LIN {X 0,Y 411.211,Z 404.262,A -85,B 0,C 180,E1 -10479.728,E2 -10479.728} C_VEL
LIN {X 0,Y 411.171,Z 404.269,A -85,B 0,C 180,E1 -10483.134,E2 -10483.134} C_VEL
LIN {X 0,Y 411.171,Z 404.27,A -85,B 0,C 180,E1 -10485.881,E2 -10485.881} C_VEL
LIN {X 0,Y 411.213,Z 404.285,A -85,B 0,C 180,E1 -10487.705,E2 -10487.705} C_VEL
LIN {X 0,Y 411.99,Z 408.991,A -85,B 0,C 180,E1 -10490.864,E2 -10490.864} C_VEL
LIN {X 0,Y 412.564,Z 413.025,A -85,B 0,C 180,E1 -10493.401,E2 -10493.401} C_VEL
LIN {X 0,Y 412.538,Z 417.134,A -85,B 0,C 180,E1 -10495.793,E2 -10495.793} C_VEL
LIN {X 0,Y 412.031,Z 423.342,A -85,B 0,C 180,E1 -10499.223,E2 -10499.223} C_VEL
LIN {X 0,Y 411.473,Z 429.833,A -85,B 0,C 180,E1 -10502.644,E2 -10502.644} C_VEL
LIN {X 0,Y 411.104,Z 435.991,A -85,B 0,C 180,E1 -10505.777,E2 -10505.777} C_VEL
LIN {X 0,Y 410.797,Z 442.38,A -85,B 0,C 180,E1 -10508.945,E2 -10508.945} C_VEL
LIN {X 0,Y 410.522,Z 449.14,A -85,B 0,C 180,E1 -10512.118,E2 -10512.118} C_VEL
LIN {X 0,Y 413.255,Z 462.27,A -85,B 0,C 180,E1 -10512.668,E2 -10512.668} C_VEL
LIN {X 0,Y 414.885,Z 474.445,A -85,B 0,C 180,E1 -10513.327,E2 -10513.327} C_VEL
LIN {X 0,Y 415.191,Z 479.769,A -85,B 0,C 180,E1 -10513.656,E2 -10513.656} C_VEL
LIN {X 0,Y 414.353,Z 492.016,A -85,B 0,C 180,E1 -10514.506,E2 -10514.506} C_VEL
LIN {X 0,Y 413.49,Z 502.748,A -85,B 0,C 180,E1 -10515.457,E2 -10515.457} C_VEL
LIN {X 0,Y 412.834,Z 511.902,A -85,B 0,C 180,E1 -10516.463,E2 -10516.463} C_VEL
LIN {X 0,Y 412.087,Z 521.077,A -85,B 0,C 180,E1 -10517.691,E2 -10517.691} C_VEL
LIN {X 0,Y 411.228,Z 530.022,A -85,B 0,C 180,E1 -10519.164,E2 -10519.164} C_VEL
LIN {X 0,Y 410.717,Z 537.242,A -85,B 0,C 180,E1 -10520.645,E2 -10520.645} C_VEL
LIN {X 0,Y 410.354,Z 543.03,A -85,B 0,C 180,E1 -10522.125,E2 -10522.125} C_VEL
LIN {X 0,Y 410.045,Z 548.033,A -85,B 0,C 180,E1 -10523.774,E2 -10523.774} C_VEL
LIN {X 0,Y 410.024,Z 551.083,A -85,B 0,C 180,E1 -10525.084,E2 -10525.084} C_VEL
LIN {X 0,Y 409.935,Z 552.834,A -85,B 0,C 180,E1 -10526.068,E2 -10526.068} C_VEL
LIN {X 0,Y 409.967,Z 555.121,A -85,B 0,C 180,E1 -10528.035,E2 -10528.035} C_VEL
LIN {X 0,Y 409.936,Z 555.676,A -85,B 0,C 180,E1 -10529.017,E2 -10529.017} C_VEL
LIN {X 0,Y 409.926,Z 555.798,A -85,B 0,C 180,E1 -10530,E2 -10530} C_VEL
LIN {X 0,Y 409.967,Z 554.868,A -85,B 0,C 180,E1 -10531.965,E2 -10531.965} C_VEL
LIN {X 0,Y 409.929,Z 553.816,A -85,B 0,C 180,E1 -10532.948,E2 -10532.948} C_VEL
LIN {X 0,Y 409.935,Z 552.312,A -85,B 0,C 180,E1 -10533.932,E2 -10533.932} C_VEL
LIN {X 0,Y 410.025,Z 549.264,A -85,B 0,C 180,E1 -10535.409,E2 -10535.409} C_VEL
LIN {X 0,Y 410.167,Z 545.148,A -85,B 0,C 180,E1 -10536.888,E2 -10536.888} C_VEL
LIN {X 0,Y 410.488,Z 538.835,A -85,B 0,C 180,E1 -10538.616,E2 -10538.616} C_VEL
LIN {X 0,Y 410.916,Z 531.955,A -85,B 0,C 180,E1 -10540.096,E2 -10540.096} C_VEL
LIN {X 0,Y 411.365,Z 524.924,A -85,B 0,C 180,E1 -10541.33,E2 -10541.33} C_VEL
LIN {X 0,Y 412.025,Z 516.459,A -85,B 0,C 180,E1 -10542.561,E2 -10542.561} C_VEL
LIN {X 0,Y 412.68,Z 505.979,A -85,B 0,C 180,E1 -10543.793,E2 -10543.793} C_VEL
LIN {X 0,Y 413.431,Z 495.616,A -85,B 0,C 180,E1 -10544.772,E2 -10544.772} C_VEL
LIN {X 0,Y 414.099,Z 484.253,A -85,B 0,C 180,E1 -10545.63,E2 -10545.63} C_VEL
LIN {X 0,Y 414.498,Z 477.243,A -85,B 0,C 180,E1 -10546.056,E2 -10546.056} C_VEL
LIN {X 0,Y 412.757,Z 464.018,A -85,B 0,C 180,E1 -10546.759,E2 -10546.759} C_VEL
LIN {X 0,Y 410.638,Z 450.81,A -85,B 0,C 180,E1 -10547.267,E2 -10547.267} C_VEL
LIN {X 0,Y 410.406,Z 449.172,A -85,B 0,C 180,E1 -10547.314,E2 -10547.314} C_VEL
LIN {X 0,Y 410.705,Z 441.204,A -85,B 0,C 180,E1 -10551.06,E2 -10551.06} C_VEL
LIN {X 0,Y 410.962,Z 434.585,A -85,B 0,C 180,E1 -10554.231,E2 -10554.231} C_VEL
LIN {X 0,Y 411.272,Z 428.297,A -85,B 0,C 180,E1 -10557.302,E2 -10557.302} C_VEL
LIN {X 0,Y 411.717,Z 422.412,A -85,B 0,C 180,E1 -10560.235,E2 -10560.235} C_VEL
LIN {X 0,Y 412.033,Z 416.434,A -85,B 0,C 180,E1 -10563.302,E2 -10563.302} C_VEL
LIN {X 0,Y 412.291,Z 412.421,A -85,B 0,C 180,E1 -10565.419,E2 -10565.419} C_VEL
LIN {X 0,Y 411.848,Z 407.948,A -85,B 0,C 180,E1 -10567.902,E2 -10567.902} C_VEL
LIN {X 0,Y 411.242,Z 404.261,A -85,B 0,C 180,E1 -10570.083,E2 -10570.083} C_VEL
LIN {X 0,Y 411.215,Z 404.265,A -85,B 0,C 180,E1 -10573.127,E2 -10573.127} C_VEL
LIN {X 0,Y 411.173,Z 404.265,A -85,B 0,C 180,E1 -10575.879,E2 -10575.879} C_VEL
LIN {X 0,Y 411.16,Z 404.271,A -85,B 0,C 180,E1 -10578.771,E2 -10578.771} C_VEL
LIN {X 0,Y 411.195,Z 404.263,A -85,B 0,C 180,E1 -10582.026,E2 -10582.026} C_VEL
LIN {X 0,Y 411.201,Z 404.263,A -85,B 0,C 180,E1 -10585.666,E2 -10585.666} C_VEL
LIN {X 0,Y 411.192,Z 404.265,A -85,B 0,C 180,E1 -10589.152,E2 -10589.152} C_VEL
LIN {X 0,Y 411.253,Z 404.26,A -85,B 0,C 180,E1 -10592.522,E2 -10592.522} C_VEL
LIN {X 0,Y 411.22,Z 404.26,A -85,B 0,C 180,E1 -10595.784,E2 -10595.784} C_VEL
LIN {X 0,Y 411.189,Z 404.266,A -85,B 0,C 180,E1 -10598.965,E2 -10598.965} C_VEL
LIN {X 0,Y 411.245,Z 404.259,A -85,B 0,C 180,E1 -10602.084,E2 -10602.084} C_VEL
LIN {X 0,Y 411.251,Z 404.258,A -85,B 0,C 180,E1 -10605.147,E2 -10605.147} C_VEL
LIN {X 0,Y 411.276,Z 404.256,A -85,B 0,C 180,E1 -10608.167,E2 -10608.167} C_VEL
LIN {X 0,Y 411.474,Z 404.232,A -85,B 0,C 180,E1 -10612.146,E2 -10612.146} C_VEL
LIN {X 0,Y 411.482,Z 404.23,A -85,B 0,C 180,E1 -10614.118,E2 -10614.118} C_VEL
LIN {X 0,Y 411.506,Z 404.227,A -85,B 0,C 180,E1 -10618.042,E2 -10618.042} C_VEL
LIN {X 0,Y 411.635,Z 404.211,A -85,B 0,C 180,E1 -10620,E2 -10620} C_VEL
LIN {X 0,Y 411.46,Z 404.231,A -85,B 0,C 180,E1 -10622.937,E2 -10622.937} C_VEL
LIN {X 0,Y 411.453,Z 404.232,A -85,B 0,C 180,E1 -10626.867,E2 -10626.867} C_VEL
LIN {X 0,Y 411.286,Z 404.254,A -85,B 0,C 180,E1 -10629.839,E2 -10629.839} C_VEL
LIN {X 0,Y 411.304,Z 404.25,A -85,B 0,C 180,E1 -10633.109,E2 -10633.109} C_VEL
LIN {X 0,Y 411.249,Z 404.257,A -85,B 0,C 180,E1 -10636.889,E2 -10636.889} C_VEL
LIN {X 0,Y 411.222,Z 404.262,A -85,B 0,C 180,E1 -10639.987,E2 -10639.987} C_VEL
LIN {X 0,Y 411.196,Z 404.263,A -85,B 0,C 180,E1 -10643.148,E2 -10643.148} C_VEL
LIN {X 0,Y 411.23,Z 404.26,A -85,B 0,C 180,E1 -10646.381,E2 -10646.381} C_VEL
LIN {X 0,Y 411.204,Z 404.264,A -85,B 0,C 180,E1 -10649.712,E2 -10649.712} C_VEL
LIN {X 0,Y 411.2,Z 404.263,A -85,B 0,C 180,E1 -10653.156,E2 -10653.156} C_VEL
LIN {X 0,Y 411.189,Z 404.263,A -85,B 0,C 180,E1 -10656.554,E2 -10656.554} C_VEL
LIN {X 0,Y 411.223,Z 404.265,A -85,B 0,C 180,E1 -10659.731,E2 -10659.731} C_VEL
LIN {X 0,Y 411.226,Z 404.259,A -85,B 0,C 180,E1 -10663.127,E2 -10663.127} C_VEL
LIN {X 0,Y 411.226,Z 404.261,A -85,B 0,C 180,E1 -10665.873,E2 -10665.873} C_VEL
LIN {X 0,Y 411.205,Z 404.26,A -85,B 0,C 180,E1 -10668.765,E2 -10668.765} C_VEL
LIN {X 0,Y 411.201,Z 404.261,A -85,B 0,C 180,E1 -10672.028,E2 -10672.028} C_VEL
LIN {X 0,Y 411.203,Z 404.264,A -85,B 0,C 180,E1 -10675.667,E2 -10675.667} C_VEL
LIN {X 0,Y 411.187,Z 404.268,A -85,B 0,C 180,E1 -10679.153,E2 -10679.153} C_VEL
LIN {X 0,Y 411.257,Z 404.254,A -85,B 0,C 180,E1 -10682.523,E2 -10682.523} C_VEL
LIN {X 0,Y 411.216,Z 404.26,A -85,B 0,C 180,E1 -10685.785,E2 -10685.785} C_VEL
LIN {X 0,Y 411.119,Z 404.272,A -85,B 0,C 180,E1 -10687.909,E2 -10687.909} C_VEL
LIN {X 0,Y 411.038,Z 404.286,A -85,B 0,C 180,E1 -10688.958,E2 -10688.958} C_VEL
LIN {X 0,Y 411.028,Z 405.412,A -85,B 0,C 180,E1 -10690.122,E2 -10690.122} C_VEL
LIN {X 0,Y 410.929,Z 409.509,A -85,B 0,C 180,E1 -10693.285,E2 -10693.285} C_VEL
LIN {X 0,Y 410.805,Z 414.704,A -85,B 0,C 180,E1 -10697.199,E2 -10697.199} C_VEL
LIN {X 0,Y 410.584,Z 420.085,A -85,B 0,C 180,E1 -10701.138,E2 -10701.138} C_VEL
LIN {X 0,Y 410.621,Z 422.814,A -85,B 0,C 180,E1 -10703.119,E2 -10703.119} C_VEL
LIN {X 0,Y 410.429,Z 427.997,A -85,B 0,C 180,E1 -10706.779,E2 -10706.779} C_VEL
LIN {X 0,Y 412.935,Z 441.081,A -85,B 0,C 180,E1 -10707.302,E2 -10707.302} C_VEL
LIN {X 0,Y 414.936,Z 451.663,A -85,B 0,C 180,E1 -10707.877,E2 -10707.877} C_VEL
LIN {X 0,Y 414.296,Z 464.392,A -85,B 0,C 180,E1 -10708.664,E2 -10708.664} C_VEL
LIN {X 0,Y 413.609,Z 475.006,A -85,B 0,C 180,E1 -10709.513,E2 -10709.513} C_VEL
LIN {X 0,Y 412.859,Z 485.842,A -85,B 0,C 180,E1 -10710.61,E2 -10710.61} C_VEL
LIN {X 0,Y 412.21,Z 494.689,A -85,B 0,C 180,E1 -10711.71,E2 -10711.71} C_VEL
LIN {X 0,Y 411.455,Z 504.315,A -85,B 0,C 180,E1 -10713.182,E2 -10713.182} C_VEL
LIN {X 0,Y 410.935,Z 511.972,A -85,B 0,C 180,E1 -10714.66,E2 -10714.66} C_VEL
LIN {X 0,Y 410.607,Z 518.371,A -85,B 0,C 180,E1 -10716.209,E2 -10716.209} C_VEL
LIN {X 0,Y 410.256,Z 523.742,A -85,B 0,C 180,E1 -10717.877,E2 -10717.877} C_VEL
LIN {X 0,Y 410.049,Z 527.342,A -85,B 0,C 180,E1 -10719.371,E2 -10719.371} C_VEL
LIN {X 0,Y 409.956,Z 529.338,A -85,B 0,C 180,E1 -10720.511,E2 -10720.511} C_VEL
LIN {X 0,Y 409.264,Z 530.53,A -85,B 0,C 180,E1 -10721.315,E2 -10721.315} C_VEL
LIN {X 0,Y 406.302,Z 531.836,A -85,B 0,C 180,E1 -10722.632,E2 -10722.632} C_VEL
LIN {X 0,Y 403.811,Z 532.355,A -85,B 0,C 180,E1 -10723.704,E2 -10723.704} C_VEL
LIN {X 0,Y 402.763,Z 532.438,A -85,B 0,C 180,E1 -10724.536,E2 -10724.536} C_VEL
LIN {X 0,Y 402.69,Z 532.364,A -85,B 0,C 180,E1 -10724.818,E2 -10724.818} C_VEL
LIN {X 0,Y 402.765,Z 531.637,A -85,B 0,C 180,E1 -10726.319,E2 -10726.319} C_VEL
LIN {X 0,Y 402.899,Z 529.294,A -85,B 0,C 180,E1 -10728.299,E2 -10728.299} C_VEL
LIN {X 0,Y 403.167,Z 526.562,A -85,B 0,C 180,E1 -10729.725,E2 -10729.725} C_VEL
LIN {X 0,Y 403.5,Z 522.035,A -85,B 0,C 180,E1 -10731.455,E2 -10731.455} C_VEL
LIN {X 0,Y 404.058,Z 515.464,A -85,B 0,C 180,E1 -10733.311,E2 -10733.311} C_VEL
LIN {X 0,Y 404.681,Z 508.327,A -85,B 0,C 180,E1 -10734.883,E2 -10734.883} C_VEL
LIN {X 0,Y 405.391,Z 500.677,A -85,B 0,C 180,E1 -10736.236,E2 -10736.236} C_VEL
LIN {X 0,Y 406.193,Z 491.422,A -85,B 0,C 180,E1 -10737.57,E2 -10737.57} C_VEL
LIN {X 0,Y 407.089,Z 481.869,A -85,B 0,C 180,E1 -10738.686,E2 -10738.686} C_VEL
LIN {X 0,Y 407.925,Z 471.292,A -85,B 0,C 180,E1 -10739.691,E2 -10739.691} C_VEL
LIN {X 0,Y 408.762,Z 459.381,A -85,B 0,C 180,E1 -10740.573,E2 -10740.573} C_VEL
LIN {X 0,Y 409.008,Z 453.009,A -85,B 0,C 180,E1 -10740.961,E2 -10740.961} C_VEL
LIN {X 0,Y 406.66,Z 441.02,A -85,B 0,C 180,E1 -10741.685,E2 -10741.685} C_VEL
LIN {X 0,Y 403.291,Z 428.389,A -85,B 0,C 180,E1 -10742.323,E2 -10742.323} C_VEL
LIN {X 0,Y 403.46,Z 423.131,A -85,B 0,C 180,E1 -10746.317,E2 -10746.317} C_VEL
LIN {X 0,Y 403.621,Z 419.902,A -85,B 0,C 180,E1 -10748.817,E2 -10748.817} C_VEL
LIN {X 0,Y 403.788,Z 416.481,A -85,B 0,C 180,E1 -10751.546,E2 -10751.546} C_VEL
LIN {X 0,Y 403.953,Z 412.879,A -85,B 0,C 180,E1 -10754.494,E2 -10754.494} C_VEL
LIN {X 0,Y 404.163,Z 409.553,A -85,B 0,C 180,E1 -10757.299,E2 -10757.299} C_VEL
LIN {X 0,Y 404.226,Z 406.491,A -85,B 0,C 180,E1 -10759.962,E2 -10759.962} C_VEL
LIN {X 0,Y 404.131,Z 405.148,A -85,B 0,C 180,E1 -10761.241,E2 -10761.241} C_VEL
LIN {X 0,Y 404.181,Z 405.145,A -85,B 0,C 180,E1 -10764.984,E2 -10764.984} C_VEL
LIN {X 0,Y 404.144,Z 405.146,A -85,B 0,C 180,E1 -10768.554,E2 -10768.554} C_VEL
LIN {X 0,Y 404.193,Z 405.137,A -85,B 0,C 180,E1 -10772,E2 -10772} C_VEL
LIN {X 0,Y 404.169,Z 405.142,A -85,B 0,C 180,E1 -10775.334,E2 -10775.334} C_VEL
LIN {X 0,Y 404.132,Z 405.145,A -85,B 0,C 180,E1 -10778.58,E2 -10778.58} C_VEL
LIN {X 0,Y 404.204,Z 405.138,A -85,B 0,C 180,E1 -10781.762,E2 -10781.762} C_VEL
LIN {X 0,Y 404.2,Z 405.137,A -85,B 0,C 180,E1 -10784.882,E2 -10784.882} C_VEL
LIN {X 0,Y 404.251,Z 405.13,A -85,B 0,C 180,E1 -10787.958,E2 -10787.958} C_VEL
LIN {X 0,Y 404.427,Z 405.11,A -85,B 0,C 180,E1 -10792.1,E2 -10792.1} C_VEL
LIN {X 0,Y 404.418,Z 405.11,A -85,B 0,C 180,E1 -10794.015,E2 -10794.015} C_VEL
LIN {X 0,Y 404.477,Z 405.104,A -85,B 0,C 180,E1 -10798.009,E2 -10798.009} C_VEL
LIN {X 0,Y 404.605,Z 405.086,A -85,B 0,C 180,E1 -10800,E2 -10800} C_VEL
LIN {X 0,Y 404.419,Z 405.109,A -85,B 0,C 180,E1 -10802.989,E2 -10802.989} C_VEL
LIN {X 0,Y 404.401,Z 405.109,A -85,B 0,C 180,E1 -10806.988,E2 -10806.988} C_VEL
LIN {X 0,Y 404.266,Z 405.13,A -85,B 0,C 180,E1 -10810.012,E2 -10810.012} C_VEL
LIN {X 0,Y 404.261,Z 405.13,A -85,B 0,C 180,E1 -10813.212,E2 -10813.212} C_VEL
LIN {X 0,Y 404.214,Z 405.136,A -85,B 0,C 180,E1 -10817.009,E2 -10817.009} C_VEL
LIN {X 0,Y 404.159,Z 405.146,A -85,B 0,C 180,E1 -10820.352,E2 -10820.352} C_VEL
LIN {X 0,Y 404.165,Z 405.144,A -85,B 0,C 180,E1 -10823.575,E2 -10823.575} C_VEL
LIN {X 0,Y 404.179,Z 405.14,A -85,B 0,C 180,E1 -10825.767,E2 -10825.767} C_VEL
LIN {X 0,Y 404.194,Z 405.14,A -85,B 0,C 180,E1 -10828,E2 -10828} C_VEL
LIN {X 0,Y 404.139,Z 405.144,A -85,B 0,C 180,E1 -10831.559,E2 -10831.559} C_VEL
LIN {X 0,Y 404.182,Z 405.139,A -85,B 0,C 180,E1 -10835.017,E2 -10835.017} C_VEL
LIN {X 0,Y 404.153,Z 405.14,A -85,B 0,C 180,E1 -10838.757,E2 -10838.757} C_VEL
LIN {X 0,Y 404.12,Z 405.149,A -85,B 0,C 180,E1 -10841.6,E2 -10841.6} C_VEL
LIN {X 0,Y 404.145,Z 405.145,A -85,B 0,C 180,E1 -10844.523,E2 -10844.523} C_VEL
LIN {X 0,Y 404.184,Z 405.324,A -85,B 0,C 180,E1 -10847.444,E2 -10847.444} C_VEL
LIN {X 0,Y 404.876,Z 409.076,A -85,B 0,C 180,E1 -10850.04,E2 -10850.04} C_VEL
LIN {X 0,Y 405.507,Z 413.425,A -85,B 0,C 180,E1 -10852.868,E2 -10852.868} C_VEL
LIN {X 0,Y 405.597,Z 417.15,A -85,B 0,C 180,E1 -10855.124,E2 -10855.124} C_VEL
LIN {X 0,Y 405.078,Z 423.338,A -85,B 0,C 180,E1 -10858.635,E2 -10858.635} C_VEL
LIN {X 0,Y 404.634,Z 428.57,A -85,B 0,C 180,E1 -10861.469,E2 -10861.469} C_VEL
LIN {X 0,Y 404.116,Z 435.939,A -85,B 0,C 180,E1 -10865.331,E2 -10865.331} C_VEL
LIN {X 0,Y 403.725,Z 443.366,A -85,B 0,C 180,E1 -10869.093,E2 -10869.093} C_VEL
LIN {X 0,Y 403.452,Z 448.874,A -85,B 0,C 180,E1 -10871.74,E2 -10871.74} C_VEL
LIN {X 0,Y 406.317,Z 462.111,A -85,B 0,C 180,E1 -10872.315,E2 -10872.315} C_VEL
LIN {X 0,Y 407.968,Z 473.966,A -85,B 0,C 180,E1 -10872.971,E2 -10872.971} C_VEL
LIN {X 0,Y 408.401,Z 480.273,A -85,B 0,C 180,E1 -10873.376,E2 -10873.376} C_VEL
LIN {X 0,Y 407.55,Z 492.36,A -85,B 0,C 180,E1 -10874.241,E2 -10874.241} C_VEL
LIN {X 0,Y 406.64,Z 502.952,A -85,B 0,C 180,E1 -10875.206,E2 -10875.206} C_VEL
LIN {X 0,Y 405.934,Z 512.024,A -85,B 0,C 180,E1 -10876.228,E2 -10876.228} C_VEL
LIN {X 0,Y 405.144,Z 521.129,A -85,B 0,C 180,E1 -10877.477,E2 -10877.477} C_VEL
LIN {X 0,Y 404.224,Z 530.031,A -85,B 0,C 180,E1 -10878.974,E2 -10878.974} C_VEL
LIN {X 0,Y 403.686,Z 537.211,A -85,B 0,C 180,E1 -10880.48,E2 -10880.48} C_VEL
LIN {X 0,Y 403.299,Z 542.957,A -85,B 0,C 180,E1 -10881.986,E2 -10881.986} C_VEL
LIN {X 0,Y 402.958,Z 548.252,A -85,B 0,C 180,E1 -10883.795,E2 -10883.795} C_VEL
LIN {X 0,Y 402.937,Z 550.956,A -85,B 0,C 180,E1 -10884.997,E2 -10884.997} C_VEL
LIN {X 0,Y 402.855,Z 552.687,A -85,B 0,C 180,E1 -10885.998,E2 -10885.998} C_VEL
LIN {X 0,Y 402.865,Z 554.947,A -85,B 0,C 180,E1 -10888,E2 -10888} C_VEL
LIN {X 0,Y 402.863,Z 555.484,A -85,B 0,C 180,E1 -10889,E2 -10889} C_VEL
LIN {X 0,Y 402.851,Z 555.588,A -85,B 0,C 180,E1 -10890,E2 -10890} C_VEL
LIN {X 0,Y 402.863,Z 555.303,A -85,B 0,C 180,E1 -10890.999,E2 -10890.999} C_VEL
LIN {X 0,Y 402.88,Z 554.633,A -85,B 0,C 180,E1 -10891.999,E2 -10891.999} C_VEL
LIN {X 0,Y 402.829,Z 553.562,A -85,B 0,C 180,E1 -10893,E2 -10893} C_VEL
LIN {X 0,Y 402.855,Z 552.038,A -85,B 0,C 180,E1 -10894.001,E2 -10894.001} C_VEL
LIN {X 0,Y 402.926,Z 548.959,A -85,B 0,C 180,E1 -10895.505,E2 -10895.505} C_VEL
LIN {X 0,Y 403.081,Z 544.812,A -85,B 0,C 180,E1 -10897.01,E2 -10897.01} C_VEL
LIN {X 0,Y 403.424,Z 538.466,A -85,B 0,C 180,E1 -10898.768,E2 -10898.768} C_VEL
LIN {X 0,Y 403.862,Z 531.548,A -85,B 0,C 180,E1 -10900.274,E2 -10900.274} C_VEL
LIN {X 0,Y 404.383,Z 524.478,A -85,B 0,C 180,E1 -10901.529,E2 -10901.529} C_VEL
LIN {X 0,Y 405.033,Z 515.949,A -85,B 0,C 180,E1 -10902.781,E2 -10902.781} C_VEL
LIN {X 0,Y 405.748,Z 505.392,A -85,B 0,C 180,E1 -10904.033,E2 -10904.033} C_VEL
LIN {X 0,Y 406.593,Z 493.504,A -85,B 0,C 180,E1 -10905.155,E2 -10905.155} C_VEL
LIN {X 0,Y 407.346,Z 481.504,A -85,B 0,C 180,E1 -10906.024,E2 -10906.024} C_VEL
LIN {X 0,Y 407.408,Z 476.897,A -85,B 0,C 180,E1 -10906.308,E2 -10906.308} C_VEL
LIN {X 0,Y 405.69,Z 463.838,A -85,B 0,C 180,E1 -10907.015,E2 -10907.015} C_VEL
LIN {X 0,Y 403.618,Z 450.803,A -85,B 0,C 180,E1 -10907.524,E2 -10907.524} C_VEL
LIN {X 0,Y 403.344,Z 448.906,A -85,B 0,C 180,E1 -10907.609,E2 -10907.609} C_VEL
LIN {X 0,Y 403.656,Z 440.915,A -85,B 0,C 180,E1 -10911.446,E2 -10911.446} C_VEL
LIN {X 0,Y 403.936,Z 434.311,A -85,B 0,C 180,E1 -10914.681,E2 -10914.681} C_VEL
LIN {X 0,Y 404.287,Z 427.671,A -85,B 0,C 180,E1 -10917.992,E2 -10917.992} C_VEL
LIN {X 0,Y 404.826,Z 421.044,A -85,B 0,C 180,E1 -10921.386,E2 -10921.386} C_VEL
LIN {X 0,Y 405.197,Z 414.384,A -85,B 0,C 180,E1 -10924.915,E2 -10924.915} C_VEL
LIN {X 0,Y 405.065,Z 410.533,A -85,B 0,C 180,E1 -10927.049,E2 -10927.049} C_VEL
LIN {X 0,Y 404.217,Z 405.137,A -85,B 0,C 180,E1 -10930.206,E2 -10930.206} C_VEL
LIN {X 0,Y 404.19,Z 405.14,A -85,B 0,C 180,E1 -10933.089,E2 -10933.089} C_VEL
LIN {X 0,Y 404.152,Z 405.14,A -85,B 0,C 180,E1 -10935.926,E2 -10935.926} C_VEL
LIN {X 0,Y 404.115,Z 405.147,A -85,B 0,C 180,E1 -10938.634,E2 -10938.634} C_VEL
LIN {X 0,Y 404.152,Z 405.141,A -85,B 0,C 180,E1 -10941.491,E2 -10941.491} C_VEL
LIN {X 0,Y 404.18,Z 405.14,A -85,B 0,C 180,E1 -10944.983,E2 -10944.983} C_VEL
LIN {X 0,Y 404.14,Z 405.145,A -85,B 0,C 180,E1 -10948.553,E2 -10948.553} C_VEL
LIN {X 0,Y 404.192,Z 405.136,A -85,B 0,C 180,E1 -10952,E2 -10952} C_VEL
LIN {X 0,Y 404.17,Z 405.14,A -85,B 0,C 180,E1 -10955.334,E2 -10955.334} C_VEL
LIN {X 0,Y 404.131,Z 405.146,A -85,B 0,C 180,E1 -10958.58,E2 -10958.58} C_VEL
LIN {X 0,Y 404.202,Z 405.134,A -85,B 0,C 180,E1 -10961.761,E2 -10961.761} C_VEL
LIN {X 0,Y 404.198,Z 405.137,A -85,B 0,C 180,E1 -10964.881,E2 -10964.881} C_VEL
LIN {X 0,Y 404.248,Z 405.13,A -85,B 0,C 180,E1 -10967.958,E2 -10967.958} C_VEL
LIN {X 0,Y 404.425,Z 405.109,A -85,B 0,C 180,E1 -10972.099,E2 -10972.099} C_VEL
LIN {X 0,Y 404.428,Z 405.109,A -85,B 0,C 180,E1 -10974.015,E2 -10974.015} C_VEL
LIN {X 0,Y 404.475,Z 405.103,A -85,B 0,C 180,E1 -10978.008,E2 -10978.008} C_VEL
LIN {X 0,Y 404.605,Z 405.087,A -85,B 0,C 180,E1 -10980,E2 -10980} C_VEL
LIN {X 0,Y 404.417,Z 405.108,A -85,B 0,C 180,E1 -10982.988,E2 -10982.988} C_VEL
LIN {X 0,Y 404.404,Z 405.11,A -85,B 0,C 180,E1 -10986.987,E2 -10986.987} C_VEL
LIN {X 0,Y 404.252,Z 405.13,A -85,B 0,C 180,E1 -10990.012,E2 -10990.012} C_VEL
LIN {X 0,Y 404.258,Z 405.127,A -85,B 0,C 180,E1 -10993.211,E2 -10993.211} C_VEL
LIN {X 0,Y 404.207,Z 405.133,A -85,B 0,C 180,E1 -10997.007,E2 -10997.007} C_VEL
LIN {X 0,Y 404.156,Z 405.143,A -85,B 0,C 180,E1 -11000.352,E2 -11000.352} C_VEL
LIN {X 0,Y 404.162,Z 405.141,A -85,B 0,C 180,E1 -11003.575,E2 -11003.575} C_VEL
LIN {X 0,Y 404.176,Z 405.14,A -85,B 0,C 180,E1 -11005.767,E2 -11005.767} C_VEL
LIN {X 0,Y 404.19,Z 405.14,A -85,B 0,C 180,E1 -11008,E2 -11008} C_VEL
LIN {X 0,Y 404.139,Z 405.144,A -85,B 0,C 180,E1 -11011.56,E2 -11011.56} C_VEL
LIN {X 0,Y 404.179,Z 405.137,A -85,B 0,C 180,E1 -11015.017,E2 -11015.017} C_VEL
LIN {X 0,Y 404.158,Z 405.139,A -85,B 0,C 180,E1 -11018.756,E2 -11018.756} C_VEL
LIN {X 0,Y 404.186,Z 405.14,A -85,B 0,C 180,E1 -11021.611,E2 -11021.611} C_VEL
LIN {X 0,Y 404.196,Z 405.133,A -85,B 0,C 180,E1 -11024.531,E2 -11024.531} C_VEL
LIN {X 0,Y 404.202,Z 405.136,A -85,B 0,C 180,E1 -11027.306,E2 -11027.306} C_VEL
LIN {X 0,Y 404.164,Z 405.139,A -85,B 0,C 180,E1 -11029.956,E2 -11029.956} C_VEL
LIN {X 0,Y 404.137,Z 405.144,A -85,B 0,C 180,E1 -11033.125,E2 -11033.125} C_VEL
LIN {X 0,Y 404.142,Z 405.14,A -85,B 0,C 180,E1 -11036.188,E2 -11036.188} C_VEL
LIN {X 0,Y 404.143,Z 405.142,A -85,B 0,C 180,E1 -11039.716,E2 -11039.716} C_VEL
LIN {X 0,Y 404.194,Z 405.139,A -85,B 0,C 180,E1 -11043.124,E2 -11043.124} C_VEL
LIN {X 0,Y 404.171,Z 405.141,A -85,B 0,C 180,E1 -11045.335,E2 -11045.335} C_VEL
LIN {X 0,Y 404.128,Z 405.145,A -85,B 0,C 180,E1 -11047.506,E2 -11047.506} C_VEL
LIN {X 0,Y 404.009,Z 405.158,A -85,B 0,C 180,E1 -11048.574,E2 -11048.574} C_VEL
LIN {X 0,Y 403.97,Z 406.064,A -85,B 0,C 180,E1 -11049.96,E2 -11049.96} C_VEL
LIN {X 0,Y 403.866,Z 410.146,A -85,B 0,C 180,E1 -11053.156,E2 -11053.156} C_VEL
LIN {X 0,Y 403.748,Z 415.319,A -85,B 0,C 180,E1 -11057.106,E2 -11057.106} C_VEL
LIN {X 0,Y 403.508,Z 420.529,A -85,B 0,C 180,E1 -11060.982,E2 -11060.982} C_VEL
LIN {X 0,Y 403.559,Z 423.344,A -85,B 0,C 180,E1 -11063.052,E2 -11063.052} C_VEL
LIN {X 0,Y 403.363,Z 428.145,A -85,B 0,C 180,E1 -11066.504,E2 -11066.504} C_VEL
LIN {X 0,Y 406.235,Z 443.034,A -85,B 0,C 180,E1 -11067.136,E2 -11067.136} C_VEL
LIN {X 0,Y 407.965,Z 452.196,A -85,B 0,C 180,E1 -11067.654,E2 -11067.654} C_VEL
LIN {X 0,Y 407.431,Z 463.966,A -85,B 0,C 180,E1 -11068.394,E2 -11068.394} C_VEL
LIN {X 0,Y 406.705,Z 474.709,A -85,B 0,C 180,E1 -11069.258,E2 -11069.258} C_VEL
LIN {X 0,Y 405.954,Z 485.657,A -85,B 0,C 180,E1 -11070.372,E2 -11070.372} C_VEL
LIN {X 0,Y 405.23,Z 494.579,A -85,B 0,C 180,E1 -11071.491,E2 -11071.491} C_VEL
LIN {X 0,Y 404.448,Z 504.256,A -85,B 0,C 180,E1 -11072.988,E2 -11072.988} C_VEL
LIN {X 0,Y 403.893,Z 511.978,A -85,B 0,C 180,E1 -11074.491,E2 -11074.491} C_VEL
LIN {X 0,Y 403.572,Z 518.162,A -85,B 0,C 180,E1 -11075.998,E2 -11075.998} C_VEL
LIN {X 0,Y 403.263,Z 523.096,A -85,B 0,C 180,E1 -11077.511,E2 -11077.511} C_VEL
LIN {X 0,Y 402.996,Z 526.911,A -85,B 0,C 180,E1 -11079.03,E2 -11079.03} C_VEL
LIN {X 0,Y 402.849,Z 529.565,A -85,B 0,C 180,E1 -11080.5,E2 -11080.5} C_VEL
LIN {X 0,Y 402.812,Z 531.668,A -85,B 0,C 180,E1 -11082.299,E2 -11082.299} C_VEL
LIN {X 0,Y 402.688,Z 532.46,A -85,B 0,C 180,E1 -11084.143,E2 -11084.143} C_VEL
LIN {X 0,Y 402.69,Z 532.364,A -85,B 0,C 180,E1 -11084.818,E2 -11084.818} C_VEL
LIN {X 0,Y 402.062,Z 532.145,A -85,B 0,C 180,E1 -11085.654,E2 -11085.654} C_VEL
LIN {X 0,Y 399.272,Z 531.288,A -85,B 0,C 180,E1 -11087.012,E2 -11087.012} C_VEL
LIN {X 0,Y 396.953,Z 530.034,A -85,B 0,C 180,E1 -11088.096,E2 -11088.096} C_VEL
LIN {X 0,Y 396.029,Z 528.682,A -85,B 0,C 180,E1 -11088.922,E2 -11088.922} C_VEL
LIN {X 0,Y 395.994,Z 528.144,A -85,B 0,C 180,E1 -11089.197,E2 -11089.197} C_VEL
LIN {X 0,Y 396.289,Z 524.633,A -85,B 0,C 180,E1 -11090.774,E2 -11090.774} C_VEL
LIN {X 0,Y 396.682,Z 519.839,A -85,B 0,C 180,E1 -11092.39,E2 -11092.39} C_VEL
LIN {X 0,Y 397.245,Z 513.657,A -85,B 0,C 180,E1 -11094.011,E2 -11094.011} C_VEL
LIN {X 0,Y 397.902,Z 506.844,A -85,B 0,C 180,E1 -11095.446,E2 -11095.446} C_VEL
LIN {X 0,Y 398.793,Z 497.792,A -85,B 0,C 180,E1 -11096.987,E2 -11096.987} C_VEL
LIN {X 0,Y 399.635,Z 488.915,A -85,B 0,C 180,E1 -11098.204,E2 -11098.204} C_VEL
LIN {X 0,Y 400.692,Z 477.927,A -85,B 0,C 180,E1 -11099.413,E2 -11099.413} C_VEL
LIN {X 0,Y 401.552,Z 467.224,A -85,B 0,C 180,E1 -11100.356,E2 -11100.356} C_VEL
LIN {X 0,Y 402.342,Z 454.903,A -85,B 0,C 180,E1 -11101.199,E2 -11101.199} C_VEL
LIN {X 0,Y 399.971,Z 442.386,A -85,B 0,C 180,E1 -11101.99,E2 -11101.99} C_VEL
LIN {X 0,Y 396.213,Z 428.617,A -85,B 0,C 180,E1 -11102.716,E2 -11102.716} C_VEL
LIN {X 0,Y 396.353,Z 424.582,A -85,B 0,C 180,E1 -11105.813,E2 -11105.813} C_VEL
LIN {X 0,Y 396.58,Z 420.845,A -85,B 0,C 180,E1 -11108.763,E2 -11108.763} C_VEL
LIN {X 0,Y 396.789,Z 416.465,A -85,B 0,C 180,E1 -11112.303,E2 -11112.303} C_VEL
LIN {X 0,Y 396.948,Z 413.152,A -85,B 0,C 180,E1 -11115.088,E2 -11115.088} C_VEL
LIN {X 0,Y 397.158,Z 409.756,A -85,B 0,C 180,E1 -11118.005,E2 -11118.005} C_VEL
LIN {X 0,Y 397.164,Z 407.073,A -85,B 0,C 180,E1 -11120.429,E2 -11120.429} C_VEL
LIN {X 0,Y 397.088,Z 406.026,A -85,B 0,C 180,E1 -11121.723,E2 -11121.723} C_VEL
LIN {X 0,Y 397.121,Z 406.024,A -85,B 0,C 180,E1 -11125.506,E2 -11125.506} C_VEL
LIN {X 0,Y 397.082,Z 406.025,A -85,B 0,C 180,E1 -11129.118,E2 -11129.118} C_VEL
LIN {X 0,Y 397.19,Z 406.011,A -85,B 0,C 180,E1 -11132.61,E2 -11132.61} C_VEL
LIN {X 0,Y 397.123,Z 406.018,A -85,B 0,C 180,E1 -11135.981,E2 -11135.981} C_VEL
LIN {X 0,Y 397.133,Z 406.017,A -85,B 0,C 180,E1 -11139.705,E2 -11139.705} C_VEL
LIN {X 0,Y 397.176,Z 406.011,A -85,B 0,C 180,E1 -11142.845,E2 -11142.845} C_VEL
LIN {X 0,Y 397.223,Z 406.005,A -85,B 0,C 180,E1 -11146.703,E2 -11146.703} C_VEL
LIN {X 0,Y 397.213,Z 406.005,A -85,B 0,C 180,E1 -11149.809,E2 -11149.809} C_VEL
LIN {X 0,Y 397.358,Z 405.988,A -85,B 0,C 180,E1 -11152.888,E2 -11152.888} C_VEL
LIN {X 0,Y 397.249,Z 406.004,A -85,B 0,C 180,E1 -11154.925,E2 -11154.925} C_VEL
LIN {X 0,Y 397.446,Z 405.98,A -85,B 0,C 180,E1 -11157.973,E2 -11157.973} C_VEL
LIN {X 0,Y 397.574,Z 405.962,A -85,B 0,C 180,E1 -11160,E2 -11160} C_VEL
LIN {X 0,Y 397.377,Z 405.986,A -85,B 0,C 180,E1 -11163.042,E2 -11163.042} C_VEL
LIN {X 0,Y 397.369,Z 405.987,A -85,B 0,C 180,E1 -11166.092,E2 -11166.092} C_VEL
LIN {X 0,Y 397.252,Z 406.002,A -85,B 0,C 180,E1 -11169.162,E2 -11169.162} C_VEL
LIN {X 0,Y 397.225,Z 406.005,A -85,B 0,C 180,E1 -11172.258,E2 -11172.258} C_VEL
LIN {X 0,Y 397.181,Z 406.011,A -85,B 0,C 180,E1 -11175.392,E2 -11175.392} C_VEL
LIN {X 0,Y 397.157,Z 406.016,A -85,B 0,C 180,E1 -11178.574,E2 -11178.574} C_VEL
LIN {X 0,Y 397.092,Z 406.026,A -85,B 0,C 180,E1 -11181.819,E2 -11181.819} C_VEL
LIN {X 0,Y 397.152,Z 406.017,A -85,B 0,C 180,E1 -11185.132,E2 -11185.132} C_VEL
LIN {X 0,Y 397.16,Z 406.017,A -85,B 0,C 180,E1 -11187.777,E2 -11187.777} C_VEL
LIN {X 0,Y 397.081,Z 406.026,A -85,B 0,C 180,E1 -11190.882,E2 -11190.882} C_VEL
LIN {X 0,Y 397.123,Z 406.017,A -85,B 0,C 180,E1 -11194.494,E2 -11194.494} C_VEL
LIN {X 0,Y 397.102,Z 406.016,A -85,B 0,C 180,E1 -11198.275,E2 -11198.275} C_VEL
LIN {X 0,Y 397.086,Z 406.022,A -85,B 0,C 180,E1 -11200.909,E2 -11200.909} C_VEL
LIN {X 0,Y 397.099,Z 406.022,A -85,B 0,C 180,E1 -11203.649,E2 -11203.649} C_VEL
LIN {X 0,Y 397.148,Z 406.206,A -85,B 0,C 180,E1 -11207.055,E2 -11207.055} C_VEL
LIN {X 0,Y 397.986,Z 411.139,A -85,B 0,C 180,E1 -11210.527,E2 -11210.527} C_VEL
LIN {X 0,Y 398.563,Z 415.167,A -85,B 0,C 180,E1 -11213.164,E2 -11213.164} C_VEL
LIN {X 0,Y 398.552,Z 419.229,A -85,B 0,C 180,E1 -11215.648,E2 -11215.648} C_VEL
LIN {X 0,Y 397.993,Z 425.421,A -85,B 0,C 180,E1 -11219.197,E2 -11219.197} C_VEL
LIN {X 0,Y 397.393,Z 431.679,A -85,B 0,C 180,E1 -11222.625,E2 -11222.625} C_VEL
LIN {X 0,Y 396.991,Z 437.992,A -85,B 0,C 180,E1 -11225.973,E2 -11225.973} C_VEL
LIN {X 0,Y 396.639,Z 444.351,A -85,B 0,C 180,E1 -11229.245,E2 -11229.245} C_VEL
LIN {X 0,Y 396.405,Z 448.584,A -85,B 0,C 180,E1 -11231.344,E2 -11231.344} C_VEL
LIN {X 0,Y 399.341,Z 461.728,A -85,B 0,C 180,E1 -11231.935,E2 -11231.935} C_VEL
LIN {X 0,Y 401.041,Z 473.258,A -85,B 0,C 180,E1 -11232.588,E2 -11232.588} C_VEL
LIN {X 0,Y 401.623,Z 480.807,A -85,B 0,C 180,E1 -11233.087,E2 -11233.087} C_VEL
LIN {X 0,Y 400.75,Z 492.736,A -85,B 0,C 180,E1 -11233.966,E2 -11233.966} C_VEL
LIN {X 0,Y 399.763,Z 503.342,A -85,B 0,C 180,E1 -11234.963,E2 -11234.963} C_VEL
LIN {X 0,Y 399.04,Z 512.181,A -85,B 0,C 180,E1 -11235.986,E2 -11235.986} C_VEL
LIN {X 0,Y 398.203,Z 521.225,A -85,B 0,C 180,E1 -11237.255,E2 -11237.255} C_VEL
LIN {X 0,Y 397.232,Z 530.068,A -85,B 0,C 180,E1 -11238.778,E2 -11238.778} C_VEL
LIN {X 0,Y 396.671,Z 537.19,A -85,B 0,C 180,E1 -11240.31,E2 -11240.31} C_VEL
LIN {X 0,Y 396.243,Z 542.887,A -85,B 0,C 180,E1 -11241.843,E2 -11241.843} C_VEL
LIN {X 0,Y 395.956,Z 547.391,A -85,B 0,C 180,E1 -11243.375,E2 -11243.375} C_VEL
LIN {X 0,Y 395.85,Z 550.826,A -85,B 0,C 180,E1 -11244.907,E2 -11244.907} C_VEL
LIN {X 0,Y 395.778,Z 552.54,A -85,B 0,C 180,E1 -11245.927,E2 -11245.927} C_VEL
LIN {X 0,Y 395.763,Z 554.774,A -85,B 0,C 180,E1 -11247.964,E2 -11247.964} C_VEL
LIN {X 0,Y 395.791,Z 555.289,A -85,B 0,C 180,E1 -11248.982,E2 -11248.982} C_VEL
LIN {X 0,Y 395.792,Z 555.08,A -85,B 0,C 180,E1 -11251.017,E2 -11251.017} C_VEL
LIN {X 0,Y 395.778,Z 554.396,A -85,B 0,C 180,E1 -11252.035,E2 -11252.035} C_VEL
LIN {X 0,Y 395.732,Z 553.304,A -85,B 0,C 180,E1 -11253.054,E2 -11253.054} C_VEL
LIN {X 0,Y 395.778,Z 551.762,A -85,B 0,C 180,E1 -11254.073,E2 -11254.073} C_VEL
LIN {X 0,Y 395.831,Z 548.144,A -85,B 0,C 180,E1 -11255.811,E2 -11255.811} C_VEL
LIN {X 0,Y 396.077,Z 542.848,A -85,B 0,C 180,E1 -11257.647,E2 -11257.647} C_VEL
LIN {X 0,Y 396.494,Z 535.933,A -85,B 0,C 180,E1 -11259.436,E2 -11259.436} C_VEL
LIN {X 0,Y 396.996,Z 528.428,A -85,B 0,C 180,E1 -11260.97,E2 -11260.97} C_VEL
LIN {X 0,Y 397.675,Z 520.771,A -85,B 0,C 180,E1 -11262.243,E2 -11262.243} C_VEL
LIN {X 0,Y 398.364,Z 511.845,A -85,B 0,C 180,E1 -11263.47,E2 -11263.47} C_VEL
LIN {X 0,Y 399.061,Z 501.084,A -85,B 0,C 180,E1 -11264.664,E2 -11264.664} C_VEL
LIN {X 0,Y 399.928,Z 489.58,A -85,B 0,C 180,E1 -11265.675,E2 -11265.675} C_VEL
LIN {X 0,Y 400.491,Z 477.937,A -85,B 0,C 180,E1 -11266.477,E2 -11266.477} C_VEL
LIN {X 0,Y 398.787,Z 464.603,A -85,B 0,C 180,E1 -11267.227,E2 -11267.227} C_VEL
LIN {X 0,Y 396.661,Z 451.376,A -85,B 0,C 180,E1 -11267.769,E2 -11267.769} C_VEL
LIN {X 0,Y 396.247,Z 448.799,A -85,B 0,C 180,E1 -11267.848,E2 -11267.848} C_VEL
LIN {X 0,Y 396.567,Z 441.743,A -85,B 0,C 180,E1 -11271.303,E2 -11271.303} C_VEL
LIN {X 0,Y 396.878,Z 435.13,A -85,B 0,C 180,E1 -11274.591,E2 -11274.591} C_VEL
LIN {X 0,Y 397.207,Z 428.849,A -85,B 0,C 180,E1 -11277.788,E2 -11277.788} C_VEL
LIN {X 0,Y 397.645,Z 422.988,A -85,B 0,C 180,E1 -11280.833,E2 -11280.833} C_VEL
LIN {X 0,Y 398.11,Z 416.342,A -85,B 0,C 180,E1 -11284.395,E2 -11284.395} C_VEL
LIN {X 0,Y 398.168,Z 412.992,A -85,B 0,C 180,E1 -11286.254,E2 -11286.254} C_VEL
LIN {X 0,Y 397.575,Z 408.393,A -85,B 0,C 180,E1 -11288.94,E2 -11288.94} C_VEL
LIN {X 0,Y 397.162,Z 406.015,A -85,B 0,C 180,E1 -11290.455,E2 -11290.455} C_VEL
LIN {X 0,Y 397.156,Z 406.012,A -85,B 0,C 180,E1 -11293.64,E2 -11293.64} C_VEL
LIN {X 0,Y 397.102,Z 406.019,A -85,B 0,C 180,E1 -11296.52,E2 -11296.52} C_VEL
LIN {X 0,Y 397.11,Z 406.018,A -85,B 0,C 180,E1 -11300.422,E2 -11300.422} C_VEL
LIN {X 0,Y 397.104,Z 406.018,A -85,B 0,C 180,E1 -11304.265,E2 -11304.265} C_VEL
LIN {X 0,Y 397.109,Z 406.022,A -85,B 0,C 180,E1 -11306.726,E2 -11306.726} C_VEL
LIN {X 0,Y 397.127,Z 406.016,A -85,B 0,C 180,E1 -11310.296,E2 -11310.296} C_VEL
LIN {X 0,Y 397.188,Z 406.012,A -85,B 0,C 180,E1 -11312.609,E2 -11312.609} C_VEL
LIN {X 0,Y 397.126,Z 406.016,A -85,B 0,C 180,E1 -11315.981,E2 -11315.981} C_VEL
LIN {X 0,Y 397.131,Z 406.015,A -85,B 0,C 180,E1 -11319.704,E2 -11319.704} C_VEL
LIN {X 0,Y 397.174,Z 406.012,A -85,B 0,C 180,E1 -11322.844,E2 -11322.844} C_VEL
LIN {X 0,Y 397.221,Z 406.006,A -85,B 0,C 180,E1 -11326.702,E2 -11326.702} C_VEL
LIN {X 0,Y 397.21,Z 406.006,A -85,B 0,C 180,E1 -11329.809,E2 -11329.809} C_VEL
LIN {X 0,Y 397.356,Z 405.989,A -85,B 0,C 180,E1 -11332.888,E2 -11332.888} C_VEL
LIN {X 0,Y 397.253,Z 406.002,A -85,B 0,C 180,E1 -11334.925,E2 -11334.925} C_VEL
LIN {X 0,Y 397.444,Z 405.979,A -85,B 0,C 180,E1 -11337.973,E2 -11337.973} C_VEL
LIN {X 0,Y 397.574,Z 405.963,A -85,B 0,C 180,E1 -11340,E2 -11340} C_VEL
LIN {X 0,Y 397.376,Z 405.985,A -85,B 0,C 180,E1 -11343.041,E2 -11343.041} C_VEL
LIN {X 0,Y 397.356,Z 405.987,A -85,B 0,C 180,E1 -11347.112,E2 -11347.112} C_VEL
LIN {X 0,Y 397.212,Z 406.008,A -85,B 0,C 180,E1 -11350.191,E2 -11350.191} C_VEL
LIN {X 0,Y 397.218,Z 406.004,A -85,B 0,C 180,E1 -11353.321,E2 -11353.321} C_VEL
LIN {X 0,Y 397.173,Z 406.01,A -85,B 0,C 180,E1 -11357.155,E2 -11357.155} C_VEL
LIN {X 0,Y 397.095,Z 406.02,A -85,B 0,C 180,E1 -11360.73,E2 -11360.73} C_VEL
LIN {X 0,Y 397.125,Z 406.02,A -85,B 0,C 180,E1 -11364.019,E2 -11364.019} C_VEL
LIN {X 0,Y 397.187,Z 406.009,A -85,B 0,C 180,E1 -11367.39,E2 -11367.39} C_VEL
LIN {X 0,Y 397.079,Z 406.021,A -85,B 0,C 180,E1 -11370.882,E2 -11370.882} C_VEL
LIN {X 0,Y 397.119,Z 406.016,A -85,B 0,C 180,E1 -11374.494,E2 -11374.494} C_VEL
LIN {X 0,Y 397.104,Z 406.018,A -85,B 0,C 180,E1 -11378.275,E2 -11378.275} C_VEL
LIN {X 0,Y 397.151,Z 406.014,A -85,B 0,C 180,E1 -11381.994,E2 -11381.994} C_VEL
LIN {X 0,Y 397.145,Z 406.013,A -85,B 0,C 180,E1 -11385.06,E2 -11385.06} C_VEL
LIN {X 0,Y 397.151,Z 406.012,A -85,B 0,C 180,E1 -11388.007,E2 -11388.007} C_VEL
LIN {X 0,Y 397.106,Z 406.02,A -85,B 0,C 180,E1 -11391.727,E2 -11391.727} C_VEL
LIN {X 0,Y 397.123,Z 406.019,A -85,B 0,C 180,E1 -11395.507,E2 -11395.507} C_VEL
LIN {X 0,Y 397.076,Z 406.025,A -85,B 0,C 180,E1 -11399.118,E2 -11399.118} C_VEL
LIN {X 0,Y 397.192,Z 406.007,A -85,B 0,C 180,E1 -11402.611,E2 -11402.611} C_VEL
LIN {X 0,Y 397.123,Z 406.015,A -85,B 0,C 180,E1 -11405.982,E2 -11405.982} C_VEL
LIN {X 0,Y 396.91,Z 406.063,A -85,B 0,C 180,E1 -11409.26,E2 -11409.26} C_VEL
LIN {X 0,Y 396.826,Z 410.084,A -85,B 0,C 180,E1 -11412.478,E2 -11412.478} C_VEL
LIN {X 0,Y 396.656,Z 414.148,A -85,B 0,C 180,E1 -11415.638,E2 -11415.638} C_VEL
LIN {X 0,Y 396.647,Z 416.863,A -85,B 0,C 180,E1 -11417.724,E2 -11417.724} C_VEL
LIN {X 0,Y 396.427,Z 422.359,A -85,B 0,C 180,E1 -11421.847,E2 -11421.847} C_VEL
LIN {X 0,Y 396.409,Z 425.129,A -85,B 0,C 180,E1 -11423.894,E2 -11423.894} C_VEL
LIN {X 0,Y 396.346,Z 428.547,A -85,B 0,C 180,E1 -11426.251,E2 -11426.251} C_VEL
LIN {X 0,Y 398.869,Z 441.61,A -85,B 0,C 180,E1 -11426.796,E2 -11426.796} C_VEL
LIN {X 0,Y 401.074,Z 454.009,A -85,B 0,C 180,E1 -11427.506,E2 -11427.506} C_VEL
LIN {X 0,Y 400.448,Z 465.218,A -85,B 0,C 180,E1 -11428.24,E2 -11428.24} C_VEL
LIN {X 0,Y 399.627,Z 477.03,A -85,B 0,C 180,E1 -11429.244,E2 -11429.244} C_VEL
LIN {X 0,Y 398.837,Z 487.577,A -85,B 0,C 180,E1 -11430.379,E2 -11430.379} C_VEL
LIN {X 0,Y 398.134,Z 496.213,A -85,B 0,C 180,E1 -11431.517,E2 -11431.517} C_VEL
LIN {X 0,Y 397.464,Z 504.175,A -85,B 0,C 180,E1 -11432.787,E2 -11432.787} C_VEL
LIN {X 0,Y 396.862,Z 511.974,A -85,B 0,C 180,E1 -11434.316,E2 -11434.316} C_VEL
LIN {X 0,Y 396.51,Z 517.281,A -85,B 0,C 180,E1 -11435.594,E2 -11435.594} C_VEL
LIN {X 0,Y 396.236,Z 522.448,A -85,B 0,C 180,E1 -11437.132,E2 -11437.132} C_VEL
LIN {X 0,Y 395.979,Z 526.473,A -85,B 0,C 180,E1 -11438.677,E2 -11438.677} C_VEL
LIN {X 0,Y 395.775,Z 529.45,A -85,B 0,C 180,E1 -11440.229,E2 -11440.229} C_VEL
LIN {X 0,Y 395.737,Z 530.864,A -85,B 0,C 180,E1 -11441.265,E2 -11441.265} C_VEL
LIN {X 0,Y 395.708,Z 531.911,A -85,B 0,C 180,E1 -11442.358,E2 -11442.358} C_VEL
LIN {X 0,Y 395.617,Z 532.484,A -85,B 0,C 180,E1 -11443.352,E2 -11443.352} C_VEL
LIN {X 0,Y 395.59,Z 532.571,A -85,B 0,C 180,E1 -11444.823,E2 -11444.823} C_VEL
LIN {X 0,Y 395.674,Z 531.759,A -85,B 0,C 180,E1 -11446.51,E2 -11446.51} C_VEL
LIN {X 0,Y 395.76,Z 530.688,A -85,B 0,C 180,E1 -11447.571,E2 -11447.571} C_VEL
LIN {X 0,Y 395.994,Z 528.144,A -85,B 0,C 180,E1 -11449.197,E2 -11449.197} C_VEL
LIN {X 0,Y 395.488,Z 526.514,A -85,B 0,C 180,E1 -11450.014,E2 -11450.014} C_VEL
LIN {X 0,Y 392.926,Z 523.462,A -85,B 0,C 180,E1 -11451.337,E2 -11451.337} C_VEL
LIN {X 0,Y 390.409,Z 519.835,A -85,B 0,C 180,E1 -11452.639,E2 -11452.639} C_VEL
LIN {X 0,Y 389.978,Z 517.15,A -85,B 0,C 180,E1 -11453.411,E2 -11453.411} C_VEL
LIN {X 0,Y 390.614,Z 510.439,A -85,B 0,C 180,E1 -11455.012,E2 -11455.012} C_VEL
LIN {X 0,Y 391.548,Z 501.756,A -85,B 0,C 180,E1 -11456.662,E2 -11456.662} C_VEL
LIN {X 0,Y 392.519,Z 491.629,A -85,B 0,C 180,E1 -11458.179,E2 -11458.179} C_VEL
LIN {X 0,Y 393.606,Z 481.355,A -85,B 0,C 180,E1 -11459.407,E2 -11459.407} C_VEL
LIN {X 0,Y 394.513,Z 471.456,A -85,B 0,C 180,E1 -11460.363,E2 -11460.363} C_VEL
LIN {X 0,Y 395.368,Z 460.11,A -85,B 0,C 180,E1 -11461.233,E2 -11461.233} C_VEL
LIN {X 0,Y 395.634,Z 456.035,A -85,B 0,C 180,E1 -11461.497,E2 -11461.497} C_VEL
LIN {X 0,Y 393.385,Z 444.168,A -85,B 0,C 180,E1 -11462.287,E2 -11462.287} C_VEL
LIN {X 0,Y 389.848,Z 431.428,A -85,B 0,C 180,E1 -11462.989,E2 -11462.989} C_VEL
LIN {X 0,Y 389.167,Z 428.822,A -85,B 0,C 180,E1 -11463.122,E2 -11463.122} C_VEL
LIN {X 0,Y 389.363,Z 424.446,A -85,B 0,C 180,E1 -11466.558,E2 -11466.558} C_VEL
LIN {X 0,Y 389.557,Z 421.216,A -85,B 0,C 180,E1 -11469.155,E2 -11469.155} C_VEL
LIN {X 0,Y 389.768,Z 417.371,A -85,B 0,C 180,E1 -11472.33,E2 -11472.33} C_VEL
LIN {X 0,Y 389.997,Z 412.949,A -85,B 0,C 180,E1 -11476.122,E2 -11476.122} C_VEL
LIN {X 0,Y 390.172,Z 409.536,A -85,B 0,C 180,E1 -11479.158,E2 -11479.158} C_VEL
LIN {X 0,Y 390.107,Z 407.65,A -85,B 0,C 180,E1 -11480.91,E2 -11480.91} C_VEL
LIN {X 0,Y 390.036,Z 406.907,A -85,B 0,C 180,E1 -11482.45,E2 -11482.45} C_VEL
LIN {X 0,Y 390.064,Z 406.902,A -85,B 0,C 180,E1 -11485.975,E2 -11485.975} C_VEL
LIN {X 0,Y 390.025,Z 406.905,A -85,B 0,C 180,E1 -11488.496,E2 -11488.496} C_VEL
LIN {X 0,Y 390.112,Z 406.892,A -85,B 0,C 180,E1 -11492.07,E2 -11492.07} C_VEL
LIN {X 0,Y 390.072,Z 406.898,A -85,B 0,C 180,E1 -11495.519,E2 -11495.519} C_VEL
LIN {X 0,Y 390.05,Z 406.901,A -85,B 0,C 180,E1 -11498.878,E2 -11498.878} C_VEL
LIN {X 0,Y 390.122,Z 406.889,A -85,B 0,C 180,E1 -11502.167,E2 -11502.167} C_VEL
LIN {X 0,Y 390.138,Z 406.886,A -85,B 0,C 180,E1 -11505.393,E2 -11505.393} C_VEL
LIN {X 0,Y 390.143,Z 406.886,A -85,B 0,C 180,E1 -11508.571,E2 -11508.571} C_VEL
LIN {X 0,Y 390.338,Z 406.864,A -85,B 0,C 180,E1 -11511.993,E2 -11511.993} C_VEL
LIN {X 0,Y 390.221,Z 406.879,A -85,B 0,C 180,E1 -11514.834,E2 -11514.834} C_VEL
LIN {X 0,Y 390.415,Z 406.855,A -85,B 0,C 180,E1 -11517.937,E2 -11517.937} C_VEL
LIN {X 0,Y 390.544,Z 406.838,A -85,B 0,C 180,E1 -11520,E2 -11520} C_VEL
LIN {X 0,Y 390.311,Z 406.866,A -85,B 0,C 180,E1 -11523.097,E2 -11523.097} C_VEL
LIN {X 0,Y 390.323,Z 406.864,A -85,B 0,C 180,E1 -11526.202,E2 -11526.202} C_VEL
LIN {X 0,Y 390.205,Z 406.88,A -85,B 0,C 180,E1 -11529.329,E2 -11529.329} C_VEL
LIN {X 0,Y 390.174,Z 406.883,A -85,B 0,C 180,E1 -11532.483,E2 -11532.483} C_VEL
LIN {X 0,Y 390.14,Z 406.889,A -85,B 0,C 180,E1 -11535.677,E2 -11535.677} C_VEL
LIN {X 0,Y 390.101,Z 406.896,A -85,B 0,C 180,E1 -11538.923,E2 -11538.923} C_VEL
LIN {X 0,Y 390.035,Z 406.904,A -85,B 0,C 180,E1 -11542.235,E2 -11542.235} C_VEL
LIN {X 0,Y 390.115,Z 406.892,A -85,B 0,C 180,E1 -11545.744,E2 -11545.744} C_VEL
LIN {X 0,Y 390.062,Z 406.899,A -85,B 0,C 180,E1 -11549.11,E2 -11549.11} C_VEL
LIN {X 0,Y 390.04,Z 406.902,A -85,B 0,C 180,E1 -11552.722,E2 -11552.722} C_VEL
LIN {X 0,Y 390.054,Z 406.897,A -85,B 0,C 180,E1 -11555.826,E2 -11555.826} C_VEL
LIN {X 0,Y 390.068,Z 406.894,A -85,B 0,C 180,E1 -11559.219,E2 -11559.219} C_VEL
LIN {X 0,Y 390.04,Z 406.902,A -85,B 0,C 180,E1 -11562.375,E2 -11562.375} C_VEL
LIN {X 0,Y 390.045,Z 406.9,A -85,B 0,C 180,E1 -11565.355,E2 -11565.355} C_VEL
LIN {X 0,Y 390.111,Z 407.051,A -85,B 0,C 180,E1 -11566.63,E2 -11566.63} C_VEL
LIN {X 0,Y 390.823,Z 411.209,A -85,B 0,C 180,E1 -11569.657,E2 -11569.657} C_VEL
LIN {X 0,Y 391.553,Z 416.208,A -85,B 0,C 180,E1 -11573.038,E2 -11573.038} C_VEL
LIN {X 0,Y 391.529,Z 420.434,A -85,B 0,C 180,E1 -11575.661,E2 -11575.661} C_VEL
LIN {X 0,Y 391.062,Z 425.424,A -85,B 0,C 180,E1 -11578.589,E2 -11578.589} C_VEL
LIN {X 0,Y 390.46,Z 431.269,A -85,B 0,C 180,E1 -11581.881,E2 -11581.881} C_VEL
LIN {X 0,Y 389.99,Z 437.958,A -85,B 0,C 180,E1 -11585.514,E2 -11585.514} C_VEL
LIN {X 0,Y 389.633,Z 444.276,A -85,B 0,C 180,E1 -11588.854,E2 -11588.854} C_VEL
LIN {X 0,Y 389.382,Z 448.466,A -85,B 0,C 180,E1 -11590.935,E2 -11590.935} C_VEL
LIN {X 0,Y 392.379,Z 461.582,A -85,B 0,C 180,E1 -11591.546,E2 -11591.546} C_VEL
LIN {X 0,Y 394.219,Z 473.762,A -85,B 0,C 180,E1 -11592.264,E2 -11592.264} C_VEL
LIN {X 0,Y 394.844,Z 481.376,A -85,B 0,C 180,E1 -11592.788,E2 -11592.788} C_VEL
LIN {X 0,Y 393.966,Z 493.094,A -85,B 0,C 180,E1 -11593.682,E2 -11593.682} C_VEL
LIN {X 0,Y 392.874,Z 503.879,A -85,B 0,C 180,E1 -11594.728,E2 -11594.728} C_VEL
LIN {X 0,Y 391.991,Z 514.281,A -85,B 0,C 180,E1 -11595.993,E2 -11595.993} C_VEL
LIN {X 0,Y 391.12,Z 522.946,A -85,B 0,C 180,E1 -11597.284,E2 -11597.284} C_VEL
LIN {X 0,Y 390.249,Z 530.114,A -85,B 0,C 180,E1 -11598.574,E2 -11598.574} C_VEL
LIN {X 0,Y 389.658,Z 537.176,A -85,B 0,C 180,E1 -11600.134,E2 -11600.134} C_VEL
LIN {X 0,Y 389.204,Z 542.831,A -85,B 0,C 180,E1 -11601.694,E2 -11601.694} C_VEL
LIN {X 0,Y 388.88,Z 547.3,A -85,B 0,C 180,E1 -11603.254,E2 -11603.254} C_VEL
LIN {X 0,Y 388.747,Z 550.702,A -85,B 0,C 180,E1 -11604.814,E2 -11604.814} C_VEL
LIN {X 0,Y 388.703,Z 552.4,A -85,B 0,C 180,E1 -11605.852,E2 -11605.852} C_VEL
LIN {X 0,Y 388.66,Z 554.604,A -85,B 0,C 180,E1 -11607.927,E2 -11607.927} C_VEL
LIN {X 0,Y 388.703,Z 555.092,A -85,B 0,C 180,E1 -11608.964,E2 -11608.964} C_VEL
LIN {X 0,Y 388.707,Z 555.166,A -85,B 0,C 180,E1 -11610,E2 -11610} C_VEL
LIN {X 0,Y 388.704,Z 554.855,A -85,B 0,C 180,E1 -11611.036,E2 -11611.036} C_VEL
LIN {X 0,Y 388.677,Z 554.157,A -85,B 0,C 180,E1 -11612.072,E2 -11612.072} C_VEL
LIN {X 0,Y 388.639,Z 553.038,A -85,B 0,C 180,E1 -11613.11,E2 -11613.11} C_VEL
LIN {X 0,Y 388.703,Z 551.479,A -85,B 0,C 180,E1 -11614.147,E2 -11614.147} C_VEL
LIN {X 0,Y 388.731,Z 548.209,A -85,B 0,C 180,E1 -11615.76,E2 -11615.76} C_VEL
LIN {X 0,Y 388.938,Z 544.126,A -85,B 0,C 180,E1 -11617.266,E2 -11617.266} C_VEL
LIN {X 0,Y 389.319,Z 537.706,A -85,B 0,C 180,E1 -11619.088,E2 -11619.088} C_VEL
LIN {X 0,Y 389.798,Z 530.694,A -85,B 0,C 180,E1 -11620.649,E2 -11620.649} C_VEL
LIN {X 0,Y 390.538,Z 521.896,A -85,B 0,C 180,E1 -11622.207,E2 -11622.207} C_VEL
LIN {X 0,Y 391.276,Z 512.876,A -85,B 0,C 180,E1 -11623.503,E2 -11623.503} C_VEL
LIN {X 0,Y 391.96,Z 502.942,A -85,B 0,C 180,E1 -11624.67,E2 -11624.67} C_VEL
LIN {X 0,Y 392.807,Z 491.954,A -85,B 0,C 180,E1 -11625.7,E2 -11625.7} C_VEL
LIN {X 0,Y 393.604,Z 479.617,A -85,B 0,C 180,E1 -11626.599,E2 -11626.599} C_VEL
LIN {X 0,Y 392.216,Z 467.913,A -85,B 0,C 180,E1 -11627.315,E2 -11627.315} C_VEL
LIN {X 0,Y 390.226,Z 454.81,A -85,B 0,C 180,E1 -11627.916,E2 -11627.916} C_VEL
LIN {X 0,Y 389.196,Z 448.555,A -85,B 0,C 180,E1 -11628.149,E2 -11628.149} C_VEL
LIN {X 0,Y 389.509,Z 441.44,A -85,B 0,C 180,E1 -11631.708,E2 -11631.708} C_VEL
LIN {X 0,Y 389.871,Z 434.854,A -85,B 0,C 180,E1 -11635.063,E2 -11635.063} C_VEL
LIN {X 0,Y 390.25,Z 428.209,A -85,B 0,C 180,E1 -11638.513,E2 -11638.513} C_VEL
LIN {X 0,Y 390.752,Z 422.718,A -85,B 0,C 180,E1 -11641.438,E2 -11641.438} C_VEL
LIN {X 0,Y 391.172,Z 416.052,A -85,B 0,C 180,E1 -11645.094,E2 -11645.094} C_VEL
LIN {X 0,Y 391.035,Z 412.724,A -85,B 0,C 180,E1 -11647.019,E2 -11647.019} C_VEL
LIN {X 0,Y 390.475,Z 408.953,A -85,B 0,C 180,E1 -11649.291,E2 -11649.291} C_VEL
LIN {X 0,Y 390.13,Z 406.891,A -85,B 0,C 180,E1 -11650.627,E2 -11650.627} C_VEL
LIN {X 0,Y 390.098,Z 406.89,A -85,B 0,C 180,E1 -11653.892,E2 -11653.892} C_VEL
LIN {X 0,Y 390.04,Z 406.899,A -85,B 0,C 180,E1 -11657.625,E2 -11657.625} C_VEL
LIN {X 0,Y 390.087,Z 406.897,A -85,B 0,C 180,E1 -11660.907,E2 -11660.907} C_VEL
LIN {X 0,Y 390.08,Z 406.897,A -85,B 0,C 180,E1 -11664.792,E2 -11664.792} C_VEL
LIN {X 0,Y 390.022,Z 406.903,A -85,B 0,C 180,E1 -11668.495,E2 -11668.495} C_VEL
LIN {X 0,Y 390.111,Z 406.889,A -85,B 0,C 180,E1 -11672.069,E2 -11672.069} C_VEL
LIN {X 0,Y 390.073,Z 406.894,A -85,B 0,C 180,E1 -11675.519,E2 -11675.519} C_VEL
LIN {X 0,Y 390.048,Z 406.9,A -85,B 0,C 180,E1 -11678.877,E2 -11678.877} C_VEL
LIN {X 0,Y 390.12,Z 406.89,A -85,B 0,C 180,E1 -11682.166,E2 -11682.166} C_VEL
LIN {X 0,Y 390.136,Z 406.886,A -85,B 0,C 180,E1 -11685.392,E2 -11685.392} C_VEL
LIN {X 0,Y 390.14,Z 406.889,A -85,B 0,C 180,E1 -11688.571,E2 -11688.571} C_VEL
LIN {X 0,Y 390.336,Z 406.863,A -85,B 0,C 180,E1 -11691.993,E2 -11691.993} C_VEL
LIN {X 0,Y 390.225,Z 406.878,A -85,B 0,C 180,E1 -11694.833,E2 -11694.833} C_VEL
LIN {X 0,Y 390.412,Z 406.854,A -85,B 0,C 180,E1 -11697.937,E2 -11697.937} C_VEL
LIN {X 0,Y 390.543,Z 406.838,A -85,B 0,C 180,E1 -11700,E2 -11700} C_VEL
LIN {X 0,Y 390.31,Z 406.865,A -85,B 0,C 180,E1 -11703.096,E2 -11703.096} C_VEL
LIN {X 0,Y 390.302,Z 406.865,A -85,B 0,C 180,E1 -11706.644,E2 -11706.644} C_VEL
LIN {X 0,Y 390.197,Z 406.879,A -85,B 0,C 180,E1 -11709.329,E2 -11709.329} C_VEL
LIN {X 0,Y 390.167,Z 406.885,A -85,B 0,C 180,E1 -11712.483,E2 -11712.483} C_VEL
LIN {X 0,Y 390.132,Z 406.889,A -85,B 0,C 180,E1 -11715.677,E2 -11715.677} C_VEL
LIN {X 0,Y 390.097,Z 406.891,A -85,B 0,C 180,E1 -11718.922,E2 -11718.922} C_VEL
LIN {X 0,Y 390.033,Z 406.902,A -85,B 0,C 180,E1 -11722.234,E2 -11722.234} C_VEL
LIN {X 0,Y 390.112,Z 406.892,A -85,B 0,C 180,E1 -11725.744,E2 -11725.744} C_VEL
LIN {X 0,Y 390.058,Z 406.896,A -85,B 0,C 180,E1 -11729.109,E2 -11729.109} C_VEL
LIN {X 0,Y 390.049,Z 406.896,A -85,B 0,C 180,E1 -11732.721,E2 -11732.721} C_VEL
LIN {X 0,Y 390.051,Z 406.901,A -85,B 0,C 180,E1 -11735.826,E2 -11735.826} C_VEL
LIN {X 0,Y 390.069,Z 406.895,A -85,B 0,C 180,E1 -11739.22,E2 -11739.22} C_VEL
LIN {X 0,Y 390.117,Z 406.888,A -85,B 0,C 180,E1 -11742.388,E2 -11742.388} C_VEL
LIN {X 0,Y 390.112,Z 406.892,A -85,B 0,C 180,E1 -11745.366,E2 -11745.366} C_VEL
LIN {X 0,Y 390.1,Z 406.89,A -85,B 0,C 180,E1 -11748.197,E2 -11748.197} C_VEL
LIN {X 0,Y 390.091,Z 406.891,A -85,B 0,C 180,E1 -11750.909,E2 -11750.909} C_VEL
LIN {X 0,Y 390.082,Z 406.892,A -85,B 0,C 180,E1 -11754.794,E2 -11754.794} C_VEL
LIN {X 0,Y 390.021,Z 406.899,A -85,B 0,C 180,E1 -11758.496,E2 -11758.496} C_VEL
LIN {X 0,Y 390.115,Z 406.888,A -85,B 0,C 180,E1 -11762.071,E2 -11762.071} C_VEL
LIN {X 0,Y 390.074,Z 406.895,A -85,B 0,C 180,E1 -11765.52,E2 -11765.52} C_VEL
LIN {X 0,Y 389.979,Z 406.906,A -85,B 0,C 180,E1 -11767.763,E2 -11767.763} C_VEL
LIN {X 0,Y 389.902,Z 406.918,A -85,B 0,C 180,E1 -11768.87,E2 -11768.87} C_VEL
LIN {X 0,Y 389.879,Z 407.801,A -85,B 0,C 180,E1 -11769.972,E2 -11769.972} C_VEL
LIN {X 0,Y 389.749,Z 411.863,A -85,B 0,C 180,E1 -11773.232,E2 -11773.232} C_VEL
LIN {X 0,Y 389.633,Z 416.541,A -85,B 0,C 180,E1 -11776.912,E2 -11776.912} C_VEL
LIN {X 0,Y 389.397,Z 421.433,A -85,B 0,C 180,E1 -11780.652,E2 -11780.652} C_VEL
LIN {X 0,Y 389.364,Z 425.574,A -85,B 0,C 180,E1 -11783.783,E2 -11783.783} C_VEL
LIN {X 0,Y 389.303,Z 428.524,A -85,B 0,C 180,E1 -11785.957,E2 -11785.957} C_VEL
LIN {X 0,Y 392.116,Z 443.469,A -85,B 0,C 180,E1 -11786.613,E2 -11786.613} C_VEL
LIN {X 0,Y 394.154,Z 455.027,A -85,B 0,C 180,E1 -11787.306,E2 -11787.306} C_VEL
LIN {X 0,Y 393.478,Z 466.411,A -85,B 0,C 180,E1 -11788.081,E2 -11788.081} C_VEL
LIN {X 0,Y 392.639,Z 477.99,A -85,B 0,C 180,E1 -11789.103,E2 -11789.103} C_VEL
LIN {X 0,Y 391.839,Z 488.405,A -85,B 0,C 180,E1 -11790.257,E2 -11790.257} C_VEL
LIN {X 0,Y 391.042,Z 497.808,A -85,B 0,C 180,E1 -11791.545,E2 -11791.545} C_VEL
LIN {X 0,Y 390.229,Z 506.877,A -85,B 0,C 180,E1 -11793.097,E2 -11793.097} C_VEL
LIN {X 0,Y 389.673,Z 514.183,A -85,B 0,C 180,E1 -11794.655,E2 -11794.655} C_VEL
LIN {X 0,Y 389.338,Z 520.035,A -85,B 0,C 180,E1 -11796.218,E2 -11796.218} C_VEL
LIN {X 0,Y 389.038,Z 524.66,A -85,B 0,C 180,E1 -11797.787,E2 -11797.787} C_VEL
LIN {X 0,Y 388.783,Z 528.188,A -85,B 0,C 180,E1 -11799.363,E2 -11799.363} C_VEL
LIN {X 0,Y 388.681,Z 529.956,A -85,B 0,C 180,E1 -11800.417,E2 -11800.417} C_VEL
LIN {X 0,Y 388.618,Z 532.156,A -85,B 0,C 180,E1 -11802.428,E2 -11802.428} C_VEL
LIN {X 0,Y 388.502,Z 532.767,A -85,B 0,C 180,E1 -11803.602,E2 -11803.602} C_VEL
LIN {X 0,Y 388.492,Z 532.847,A -85,B 0,C 180,E1 -11804.671,E2 -11804.671} C_VEL
LIN {X 0,Y 388.595,Z 532.001,A -85,B 0,C 180,E1 -11806.557,E2 -11806.557} C_VEL
LIN {X 0,Y 388.718,Z 530.606,A -85,B 0,C 180,E1 -11807.9,E2 -11807.9} C_VEL
LIN {X 0,Y 388.97,Z 527.983,A -85,B 0,C 180,E1 -11809.527,E2 -11809.527} C_VEL
LIN {X 0,Y 389.291,Z 524.252,A -85,B 0,C 180,E1 -11811.165,E2 -11811.165} C_VEL
LIN {X 0,Y 389.732,Z 519.613,A -85,B 0,C 180,E1 -11812.716,E2 -11812.716} C_VEL
LIN {X 0,Y 389.978,Z 517.15,A -85,B 0,C 180,E1 -11813.411,E2 -11813.411} C_VEL
LIN {X 0,Y 389.6,Z 514.286,A -85,B 0,C 180,E1 -11814.167,E2 -11814.167} C_VEL
LIN {X 0,Y 387.352,Z 509.338,A -85,B 0,C 180,E1 -11815.394,E2 -11815.394} C_VEL
LIN {X 0,Y 385.17,Z 503.872,A -85,B 0,C 180,E1 -11816.577,E2 -11816.577} C_VEL
LIN {X 0,Y 384.892,Z 500.109,A -85,B 0,C 180,E1 -11817.253,E2 -11817.253} C_VEL
LIN {X 0,Y 385.767,Z 491.564,A -85,B 0,C 180,E1 -11818.527,E2 -11818.527} C_VEL
LIN {X 0,Y 386.943,Z 480.872,A -85,B 0,C 180,E1 -11819.815,E2 -11819.815} C_VEL
LIN {X 0,Y 387.889,Z 470.776,A -85,B 0,C 180,E1 -11820.787,E2 -11820.787} C_VEL
LIN {X 0,Y 388.803,Z 458.859,A -85,B 0,C 180,E1 -11821.691,E2 -11821.691} C_VEL
LIN {X 0,Y 388.535,Z 454.702,A -85,B 0,C 180,E1 -11821.986,E2 -11821.986} C_VEL
LIN {X 0,Y 386.06,Z 442.964,A -85,B 0,C 180,E1 -11822.776,E2 -11822.776} C_VEL
LIN {X 0,Y 382.603,Z 431.045,A -85,B 0,C 180,E1 -11823.45,E2 -11823.45} C_VEL
LIN {X 0,Y 382.163,Z 429.017,A -85,B 0,C 180,E1 -11823.574,E2 -11823.574} C_VEL
LIN {X 0,Y 382.365,Z 424.316,A -85,B 0,C 180,E1 -11827.34,E2 -11827.34} C_VEL
LIN {X 0,Y 382.551,Z 421.073,A -85,B 0,C 180,E1 -11830.015,E2 -11830.015} C_VEL
LIN {X 0,Y 382.755,Z 417.774,A -85,B 0,C 180,E1 -11832.794,E2 -11832.794} C_VEL
LIN {X 0,Y 382.931,Z 414.364,A -85,B 0,C 180,E1 -11835.78,E2 -11835.78} C_VEL
LIN {X 0,Y 383.14,Z 411.029,A -85,B 0,C 180,E1 -11838.769,E2 -11838.769} C_VEL
LIN {X 0,Y 383.014,Z 408.268,A -85,B 0,C 180,E1 -11841.401,E2 -11841.401} C_VEL
LIN {X 0,Y 382.992,Z 407.783,A -85,B 0,C 180,E1 -11842.097,E2 -11842.097} C_VEL
LIN {X 0,Y 383.014,Z 407.782,A -85,B 0,C 180,E1 -11845.332,E2 -11845.332} C_VEL
LIN {X 0,Y 383.032,Z 407.777,A -85,B 0,C 180,E1 -11847.853,E2 -11847.853} C_VEL
LIN {X 0,Y 383.059,Z 407.77,A -85,B 0,C 180,E1 -11851.72,E2 -11851.72} C_VEL
LIN {X 0,Y 383.046,Z 407.772,A -85,B 0,C 180,E1 -11855.039,E2 -11855.039} C_VEL
LIN {X 0,Y 382.986,Z 407.778,A -85,B 0,C 180,E1 -11858.469,E2 -11858.469} C_VEL
LIN {X 0,Y 383.083,Z 407.768,A -85,B 0,C 180,E1 -11861.828,E2 -11861.828} C_VEL
LIN {X 0,Y 383.104,Z 407.763,A -85,B 0,C 180,E1 -11865.118,E2 -11865.118} C_VEL
LIN {X 0,Y 383.092,Z 407.764,A -85,B 0,C 180,E1 -11868.358,E2 -11868.358} C_VEL
LIN {X 0,Y 383.298,Z 407.741,A -85,B 0,C 180,E1 -11871.933,E2 -11871.933} C_VEL
LIN {X 0,Y 383.193,Z 407.754,A -85,B 0,C 180,E1 -11874.739,E2 -11874.739} C_VEL
LIN {X 0,Y 383.382,Z 407.731,A -85,B 0,C 180,E1 -11877.899,E2 -11877.899} C_VEL
LIN {X 0,Y 383.513,Z 407.714,A -85,B 0,C 180,E1 -11880,E2 -11880} C_VEL
LIN {X 0,Y 383.248,Z 407.746,A -85,B 0,C 180,E1 -11883.154,E2 -11883.154} C_VEL
LIN {X 0,Y 383.279,Z 407.742,A -85,B 0,C 180,E1 -11886.317,E2 -11886.317} C_VEL
LIN {X 0,Y 383.151,Z 407.759,A -85,B 0,C 180,E1 -11889.502,E2 -11889.502} C_VEL
LIN {X 0,Y 383.137,Z 407.761,A -85,B 0,C 180,E1 -11892.716,E2 -11892.716} C_VEL
LIN {X 0,Y 383.081,Z 407.77,A -85,B 0,C 180,E1 -11895.974,E2 -11895.974} C_VEL
LIN {X 0,Y 383.056,Z 407.773,A -85,B 0,C 180,E1 -11899.284,E2 -11899.284} C_VEL
LIN {X 0,Y 383.033,Z 407.777,A -85,B 0,C 180,E1 -11903.451,E2 -11903.451} C_VEL
LIN {X 0,Y 383.076,Z 407.77,A -85,B 0,C 180,E1 -11906.124,E2 -11906.124} C_VEL
LIN {X 0,Y 383.046,Z 407.772,A -85,B 0,C 180,E1 -11908.492,E2 -11908.492} C_VEL
LIN {X 0,Y 383.008,Z 407.778,A -85,B 0,C 180,E1 -11912.15,E2 -11912.15} C_VEL
LIN {X 0,Y 383.015,Z 407.775,A -85,B 0,C 180,E1 -11914.669,E2 -11914.669} C_VEL
LIN {X 0,Y 382.998,Z 407.772,A -85,B 0,C 180,E1 -11917.905,E2 -11917.905} C_VEL
LIN {X 0,Y 382.981,Z 407.781,A -85,B 0,C 180,E1 -11921.348,E2 -11921.348} C_VEL
LIN {X 0,Y 382.995,Z 407.778,A -85,B 0,C 180,E1 -11924.304,E2 -11924.304} C_VEL
LIN {X 0,Y 383.045,Z 407.881,A -85,B 0,C 180,E1 -11926.167,E2 -11926.167} C_VEL
LIN {X 0,Y 383.638,Z 411.294,A -85,B 0,C 180,E1 -11928.739,E2 -11928.739} C_VEL
LIN {X 0,Y 384.322,Z 415.707,A -85,B 0,C 180,E1 -11931.844,E2 -11931.844} C_VEL
LIN {X 0,Y 384.61,Z 419.286,A -85,B 0,C 180,E1 -11934.216,E2 -11934.216} C_VEL
LIN {X 0,Y 384.413,Z 422.342,A -85,B 0,C 180,E1 -11936.11,E2 -11936.11} C_VEL
LIN {X 0,Y 383.873,Z 427.833,A -85,B 0,C 180,E1 -11939.371,E2 -11939.371} C_VEL
LIN {X 0,Y 383.294,Z 433.712,A -85,B 0,C 180,E1 -11942.717,E2 -11942.717} C_VEL
LIN {X 0,Y 382.799,Z 440.831,A -85,B 0,C 180,E1 -11946.632,E2 -11946.632} C_VEL
LIN {X 0,Y 382.396,Z 447.365,A -85,B 0,C 180,E1 -11950.123,E2 -11950.123} C_VEL
LIN {X 0,Y 382.358,Z 448.275,A -85,B 0,C 180,E1 -11950.505,E2 -11950.505} C_VEL
LIN {X 0,Y 385.5,Z 461.803,A -85,B 0,C 180,E1 -11951.163,E2 -11951.163} C_VEL
LIN {X 0,Y 387.422,Z 473.713,A -85,B 0,C 180,E1 -11951.893,E2 -11951.893} C_VEL
LIN {X 0,Y 388.08,Z 482.009,A -85,B 0,C 180,E1 -11952.478,E2 -11952.478} C_VEL
LIN {X 0,Y 387.186,Z 493.49,A -85,B 0,C 180,E1 -11953.388,E2 -11953.388} C_VEL
LIN {X 0,Y 386.058,Z 503.938,A -85,B 0,C 180,E1 -11954.424,E2 -11954.424} C_VEL
LIN {X 0,Y 385.184,Z 513.622,A -85,B 0,C 180,E1 -11955.622,E2 -11955.622} C_VEL
LIN {X 0,Y 384.189,Z 523.062,A -85,B 0,C 180,E1 -11957.051,E2 -11957.051} C_VEL
LIN {X 0,Y 383.148,Z 531.421,A -85,B 0,C 180,E1 -11958.628,E2 -11958.628} C_VEL
LIN {X 0,Y 382.534,Z 538.169,A -85,B 0,C 180,E1 -11960.215,E2 -11960.215} C_VEL
LIN {X 0,Y 382.014,Z 544.394,A -85,B 0,C 180,E1 -11962.069,E2 -11962.069} C_VEL
LIN {X 0,Y 381.697,Z 548.914,A -85,B 0,C 180,E1 -11963.87,E2 -11963.87} C_VEL
LIN {X 0,Y 381.628,Z 552.263,A -85,B 0,C 180,E1 -11965.775,E2 -11965.775} C_VEL
LIN {X 0,Y 381.559,Z 554.435,A -85,B 0,C 180,E1 -11967.889,E2 -11967.889} C_VEL
LIN {X 0,Y 381.617,Z 554.895,A -85,B 0,C 180,E1 -11968.945,E2 -11968.945} C_VEL
LIN {X 0,Y 381.639,Z 554.955,A -85,B 0,C 180,E1 -11970,E2 -11970} C_VEL
LIN {X 0,Y 381.619,Z 554.628,A -85,B 0,C 180,E1 -11971.055,E2 -11971.055} C_VEL
LIN {X 0,Y 381.576,Z 553.914,A -85,B 0,C 180,E1 -11972.111,E2 -11972.111} C_VEL
LIN {X 0,Y 381.55,Z 552.765,A -85,B 0,C 180,E1 -11973.167,E2 -11973.167} C_VEL
LIN {X 0,Y 381.628,Z 551.191,A -85,B 0,C 180,E1 -11974.224,E2 -11974.224} C_VEL
LIN {X 0,Y 381.689,Z 547.288,A -85,B 0,C 180,E1 -11976.12,E2 -11976.12} C_VEL
LIN {X 0,Y 381.955,Z 542.118,A -85,B 0,C 180,E1 -11977.932,E2 -11977.932} C_VEL
LIN {X 0,Y 382.413,Z 535.103,A -85,B 0,C 180,E1 -11979.787,E2 -11979.787} C_VEL
LIN {X 0,Y 382.966,Z 527.502,A -85,B 0,C 180,E1 -11981.377,E2 -11981.377} C_VEL
LIN {X 0,Y 383.713,Z 519.739,A -85,B 0,C 180,E1 -11982.696,E2 -11982.696} C_VEL
LIN {X 0,Y 384.537,Z 509.813,A -85,B 0,C 180,E1 -11984.068,E2 -11984.068} C_VEL
LIN {X 0,Y 385.291,Z 499.695,A -85,B 0,C 180,E1 -11985.201,E2 -11985.201} C_VEL
LIN {X 0,Y 386.191,Z 487.958,A -85,B 0,C 180,E1 -11986.248,E2 -11986.248} C_VEL
LIN {X 0,Y 386.615,Z 479.63,A -85,B 0,C 180,E1 -11986.84,E2 -11986.84} C_VEL
LIN {X 0,Y 385,Z 466.51,A -85,B 0,C 180,E1 -11987.652,E2 -11987.652} C_VEL
LIN {X 0,Y 382.946,Z 453.22,A -85,B 0,C 180,E1 -11988.248,E2 -11988.248} C_VEL
LIN {X 0,Y 382.125,Z 448.394,A -85,B 0,C 180,E1 -11988.427,E2 -11988.427} C_VEL
LIN {X 0,Y 382.48,Z 441.138,A -85,B 0,C 180,E1 -11992.128,E2 -11992.128} C_VEL
LIN {X 0,Y 382.777,Z 435.651,A -85,B 0,C 180,E1 -11994.979,E2 -11994.979} C_VEL
LIN {X 0,Y 383.274,Z 427.944,A -85,B 0,C 180,E1 -11999.072,E2 -11999.072} C_VEL
LIN {X 0,Y 383.728,Z 422.433,A -85,B 0,C 180,E1 -12002.081,E2 -12002.081} C_VEL
LIN {X 0,Y 384.144,Z 416.889,A -85,B 0,C 180,E1 -12005.189,E2 -12005.189} C_VEL
LIN {X 0,Y 383.982,Z 413.545,A -85,B 0,C 180,E1 -12007.156,E2 -12007.156} C_VEL
LIN {X 0,Y 383.292,Z 409.072,A -85,B 0,C 180,E1 -12009.922,E2 -12009.922} C_VEL
LIN {X 0,Y 383.072,Z 407.771,A -85,B 0,C 180,E1 -12010.819,E2 -12010.819} C_VEL
LIN {X 0,Y 383.031,Z 407.77,A -85,B 0,C 180,E1 -12014.308,E2 -12014.308} C_VEL
LIN {X 0,Y 383.006,Z 407.777,A -85,B 0,C 180,E1 -12017.239,E2 -12017.239} C_VEL
LIN {X 0,Y 383.012,Z 407.774,A -85,B 0,C 180,E1 -12020.412,E2 -12020.412} C_VEL
LIN {X 0,Y 383.021,Z 407.772,A -85,B 0,C 180,E1 -12024.044,E2 -12024.044} C_VEL
LIN {X 0,Y 382.982,Z 407.777,A -85,B 0,C 180,E1 -12027.577,E2 -12027.577} C_VEL
LIN {X 0,Y 382.992,Z 407.777,A -85,B 0,C 180,E1 -12030.3,E2 -12030.3} C_VEL
LIN {X 0,Y 383.05,Z 407.773,A -85,B 0,C 180,E1 -12032.697,E2 -12032.697} C_VEL
LIN {X 0,Y 383.046,Z 407.772,A -85,B 0,C 180,E1 -12035.039,E2 -12035.039} C_VEL
LIN {X 0,Y 382.986,Z 407.78,A -85,B 0,C 180,E1 -12038.468,E2 -12038.468} C_VEL
LIN {X 0,Y 383.055,Z 407.768,A -85,B 0,C 180,E1 -12041.826,E2 -12041.826} C_VEL
LIN {X 0,Y 383.102,Z 407.764,A -85,B 0,C 180,E1 -12045.118,E2 -12045.118} C_VEL
LIN {X 0,Y 383.09,Z 407.768,A -85,B 0,C 180,E1 -12048.357,E2 -12048.357} C_VEL
LIN {X 0,Y 383.296,Z 407.739,A -85,B 0,C 180,E1 -12051.933,E2 -12051.933} C_VEL
LIN {X 0,Y 383.197,Z 407.754,A -85,B 0,C 180,E1 -12054.738,E2 -12054.738} C_VEL
LIN {X 0,Y 383.38,Z 407.729,A -85,B 0,C 180,E1 -12057.899,E2 -12057.899} C_VEL
LIN {X 0,Y 383.513,Z 407.714,A -85,B 0,C 180,E1 -12060,E2 -12060} C_VEL
LIN {X 0,Y 383.246,Z 407.744,A -85,B 0,C 180,E1 -12063.153,E2 -12063.153} C_VEL
LIN {X 0,Y 383.261,Z 407.743,A -85,B 0,C 180,E1 -12066.638,E2 -12066.638} C_VEL
LIN {X 0,Y 383.252,Z 407.747,A -85,B 0,C 180,E1 -12068.436,E2 -12068.436} C_VEL
LIN {X 0,Y 383.095,Z 407.765,A -85,B 0,C 180,E1 -12071.642,E2 -12071.642} C_VEL
LIN {X 0,Y 383.104,Z 407.762,A -85,B 0,C 180,E1 -12074.882,E2 -12074.882} C_VEL
LIN {X 0,Y 383.081,Z 407.769,A -85,B 0,C 180,E1 -12078.173,E2 -12078.173} C_VEL
LIN {X 0,Y 382.986,Z 407.778,A -85,B 0,C 180,E1 -12081.531,E2 -12081.531} C_VEL
LIN {X 0,Y 383.045,Z 407.769,A -85,B 0,C 180,E1 -12084.961,E2 -12084.961} C_VEL
LIN {X 0,Y 383.042,Z 407.77,A -85,B 0,C 180,E1 -12088.492,E2 -12088.492} C_VEL
LIN {X 0,Y 383.001,Z 407.775,A -85,B 0,C 180,E1 -12092.428,E2 -12092.428} C_VEL
LIN {X 0,Y 383.02,Z 407.776,A -85,B 0,C 180,E1 -12095.956,E2 -12095.956} C_VEL
LIN {X 0,Y 383.017,Z 407.777,A -85,B 0,C 180,E1 -12099.588,E2 -12099.588} C_VEL
LIN {X 0,Y 383.06,Z 407.766,A -85,B 0,C 180,E1 -12102.789,E2 -12102.789} C_VEL
LIN {X 0,Y 383.065,Z 407.769,A -85,B 0,C 180,E1 -12105.801,E2 -12105.801} C_VEL
LIN {X 0,Y 383.04,Z 407.769,A -85,B 0,C 180,E1 -12108.787,E2 -12108.787} C_VEL
LIN {X 0,Y 382.999,Z 407.774,A -85,B 0,C 180,E1 -12112.096,E2 -12112.096} C_VEL
LIN {X 0,Y 383.015,Z 407.778,A -85,B 0,C 180,E1 -12115.333,E2 -12115.333} C_VEL
LIN {X 0,Y 382.98,Z 407.78,A -85,B 0,C 180,E1 -12119.082,E2 -12119.082} C_VEL
LIN {X 0,Y 383.055,Z 407.768,A -85,B 0,C 180,E1 -12122.699,E2 -12122.699} C_VEL
LIN {X 0,Y 383.048,Z 407.773,A -85,B 0,C 180,E1 -12125.04,E2 -12125.04} C_VEL
LIN {X 0,Y 382.89,Z 407.788,A -85,B 0,C 180,E1 -12128.464,E2 -12128.464} C_VEL
LIN {X 0,Y 382.843,Z 408.21,A -85,B 0,C 180,E1 -12129.587,E2 -12129.587} C_VEL
LIN {X 0,Y 382.707,Z 412.26,A -85,B 0,C 180,E1 -12132.914,E2 -12132.914} C_VEL
LIN {X 0,Y 382.569,Z 417.157,A -85,B 0,C 180,E1 -12136.815,E2 -12136.815} C_VEL
LIN {X 0,Y 382.327,Z 421.865,A -85,B 0,C 180,E1 -12140.478,E2 -12140.478} C_VEL
LIN {X 0,Y 382.321,Z 426.055,A -85,B 0,C 180,E1 -12143.668,E2 -12143.668} C_VEL
LIN {X 0,Y 382.244,Z 428.748,A -85,B 0,C 180,E1 -12145.684,E2 -12145.684} C_VEL
LIN {X 0,Y 384.777,Z 441.937,A -85,B 0,C 180,E1 -12146.253,E2 -12146.253} C_VEL
LIN {X 0,Y 387.07,Z 454.452,A -85,B 0,C 180,E1 -12147,E2 -12147} C_VEL
LIN {X 0,Y 386.961,Z 461.58,A -85,B 0,C 180,E1 -12147.47,E2 -12147.47} C_VEL
LIN {X 0,Y 386.068,Z 473.556,A -85,B 0,C 180,E1 -12148.436,E2 -12148.436} C_VEL
LIN {X 0,Y 385.211,Z 484.929,A -85,B 0,C 180,E1 -12149.608,E2 -12149.608} C_VEL
LIN {X 0,Y 384.383,Z 494.106,A -85,B 0,C 180,E1 -12150.786,E2 -12150.786} C_VEL
LIN {X 0,Y 383.643,Z 502.483,A -85,B 0,C 180,E1 -12152.1,E2 -12152.1} C_VEL
LIN {X 0,Y 382.917,Z 510.677,A -85,B 0,C 180,E1 -12153.683,E2 -12153.683} C_VEL
LIN {X 0,Y 382.376,Z 517.28,A -85,B 0,C 180,E1 -12155.273,E2 -12155.273} C_VEL
LIN {X 0,Y 382.129,Z 522.058,A -85,B 0,C 180,E1 -12156.711,E2 -12156.711} C_VEL
LIN {X 0,Y 381.833,Z 526.633,A -85,B 0,C 180,E1 -12158.467,E2 -12158.467} C_VEL
LIN {X 0,Y 381.678,Z 528.768,A -85,B 0,C 180,E1 -12159.539,E2 -12159.539} C_VEL
LIN {X 0,Y 381.567,Z 530.454,A -85,B 0,C 180,E1 -12160.614,E2 -12160.614} C_VEL
LIN {X 0,Y 381.535,Z 532.404,A -85,B 0,C 180,E1 -12162.506,E2 -12162.506} C_VEL
LIN {X 0,Y 381.405,Z 533.006,A -85,B 0,C 180,E1 -12163.86,E2 -12163.86} C_VEL
LIN {X 0,Y 381.397,Z 533.022,A -85,B 0,C 180,E1 -12164.95,E2 -12164.95} C_VEL
LIN {X 0,Y 381.512,Z 532.185,A -85,B 0,C 180,E1 -12166.682,E2 -12166.682} C_VEL
LIN {X 0,Y 381.67,Z 530.514,A -85,B 0,C 180,E1 -12168.242,E2 -12168.242} C_VEL
LIN {X 0,Y 382.048,Z 527.048,A -85,B 0,C 180,E1 -12170.253,E2 -12170.253} C_VEL
LIN {X 0,Y 382.464,Z 522.312,A -85,B 0,C 180,E1 -12172.129,E2 -12172.129} C_VEL
LIN {X 0,Y 383.069,Z 516.725,A -85,B 0,C 180,E1 -12173.805,E2 -12173.805} C_VEL
LIN {X 0,Y 383.821,Z 509.635,A -85,B 0,C 180,E1 -12175.486,E2 -12175.486} C_VEL
LIN {X 0,Y 384.669,Z 502.068,A -85,B 0,C 180,E1 -12176.93,E2 -12176.93} C_VEL
LIN {X 0,Y 384.892,Z 500.109,A -85,B 0,C 180,E1 -12177.253,E2 -12177.253} C_VEL
LIN {X 0,Y 384.48,Z 497.525,A -85,B 0,C 180,E1 -12177.702,E2 -12177.702} C_VEL
LIN {X 0,Y 379.904,Z 489.273,A -85,B 0,C 180,E1 -12179.154,E2 -12179.154} C_VEL
LIN {X 0,Y 379.663,Z 486.311,A -85,B 0,C 180,E1 -12179.555,E2 -12179.555} C_VEL
LIN {X 0,Y 380.679,Z 476.224,A -85,B 0,C 180,E1 -12180.664,E2 -12180.664} C_VEL
LIN {X 0,Y 381.795,Z 464.222,A -85,B 0,C 180,E1 -12181.698,E2 -12181.698} C_VEL
LIN {X 0,Y 382.066,Z 457.255,A -85,B 0,C 180,E1 -12182.204,E2 -12182.204} C_VEL
LIN {X 0,Y 379.803,Z 445.93,A -85,B 0,C 180,E1 -12183.027,E2 -12183.027} C_VEL
LIN {X 0,Y 376.52,Z 434.109,A -85,B 0,C 180,E1 -12183.746,E2 -12183.746} C_VEL
LIN {X 0,Y 375.098,Z 429.227,A -85,B 0,C 180,E1 -12184.021,E2 -12184.021} C_VEL
LIN {X 0,Y 375.264,Z 425.791,A -85,B 0,C 180,E1 -12186.819,E2 -12186.819} C_VEL
LIN {X 0,Y 375.507,Z 422.133,A -85,B 0,C 180,E1 -12189.883,E2 -12189.883} C_VEL
LIN {X 0,Y 375.712,Z 418.322,A -85,B 0,C 180,E1 -12193.154,E2 -12193.154} C_VEL
LIN {X 0,Y 375.97,Z 414.238,A -85,B 0,C 180,E1 -12196.804,E2 -12196.804} C_VEL
LIN {X 0,Y 376.136,Z 410.811,A -85,B 0,C 180,E1 -12200.002,E2 -12200.002} C_VEL
LIN {X 0,Y 375.962,Z 408.876,A -85,B 0,C 180,E1 -12201.911,E2 -12201.911} C_VEL
LIN {X 0,Y 375.975,Z 408.659,A -85,B 0,C 180,E1 -12205.332,E2 -12205.332} C_VEL
LIN {X 0,Y 375.968,Z 408.656,A -85,B 0,C 180,E1 -12208.439,E2 -12208.439} C_VEL
LIN {X 0,Y 375.998,Z 408.65,A -85,B 0,C 180,E1 -12212.142,E2 -12212.142} C_VEL
LIN {X 0,Y 376.001,Z 408.651,A -85,B 0,C 180,E1 -12214.539,E2 -12214.539} C_VEL
LIN {X 0,Y 375.952,Z 408.654,A -85,B 0,C 180,E1 -12218.045,E2 -12218.045} C_VEL
LIN {X 0,Y 376.018,Z 408.648,A -85,B 0,C 180,E1 -12221.474,E2 -12221.474} C_VEL
LIN {X 0,Y 376.052,Z 408.643,A -85,B 0,C 180,E1 -12224.833,E2 -12224.833} C_VEL
LIN {X 0,Y 376.045,Z 408.642,A -85,B 0,C 180,E1 -12228.137,E2 -12228.137} C_VEL
LIN {X 0,Y 376.252,Z 408.618,A -85,B 0,C 180,E1 -12231.878,E2 -12231.878} C_VEL
LIN {X 0,Y 376.166,Z 408.629,A -85,B 0,C 180,E1 -12234.64,E2 -12234.64} C_VEL
LIN {X 0,Y 376.348,Z 408.607,A -85,B 0,C 180,E1 -12237.86,E2 -12237.86} C_VEL
LIN {X 0,Y 376.483,Z 408.589,A -85,B 0,C 180,E1 -12240,E2 -12240} C_VEL
LIN {X 0,Y 376.186,Z 408.625,A -85,B 0,C 180,E1 -12243.213,E2 -12243.213} C_VEL
LIN {X 0,Y 376.237,Z 408.619,A -85,B 0,C 180,E1 -12246.435,E2 -12246.435} C_VEL
LIN {X 0,Y 376.119,Z 408.635,A -85,B 0,C 180,E1 -12249.682,E2 -12249.682} C_VEL
LIN {X 0,Y 376.085,Z 408.638,A -85,B 0,C 180,E1 -12253.658,E2 -12253.658} C_VEL
LIN {X 0,Y 376.047,Z 408.646,A -85,B 0,C 180,E1 -12257.399,E2 -12257.399} C_VEL
LIN {X 0,Y 375.974,Z 408.655,A -85,B 0,C 180,E1 -12260.833,E2 -12260.833} C_VEL
LIN {X 0,Y 375.99,Z 408.652,A -85,B 0,C 180,E1 -12264.282,E2 -12264.282} C_VEL
LIN {X 0,Y 376.016,Z 408.65,A -85,B 0,C 180,E1 -12266.653,E2 -12266.653} C_VEL
LIN {X 0,Y 375.973,Z 408.654,A -85,B 0,C 180,E1 -12269.079,E2 -12269.079} C_VEL
LIN {X 0,Y 375.946,Z 408.657,A -85,B 0,C 180,E1 -12272.829,E2 -12272.829} C_VEL
LIN {X 0,Y 375.955,Z 408.654,A -85,B 0,C 180,E1 -12275.416,E2 -12275.416} C_VEL
LIN {X 0,Y 375.973,Z 408.647,A -85,B 0,C 180,E1 -12278.271,E2 -12278.271} C_VEL
LIN {X 0,Y 375.932,Z 408.66,A -85,B 0,C 180,E1 -12281.601,E2 -12281.601} C_VEL
LIN {X 0,Y 375.927,Z 408.659,A -85,B 0,C 180,E1 -12285.269,E2 -12285.269} C_VEL
LIN {X 0,Y 375.975,Z 408.821,A -85,B 0,C 180,E1 -12285.768,E2 -12285.768} C_VEL
LIN {X 0,Y 376.764,Z 413.348,A -85,B 0,C 180,E1 -12289.242,E2 -12289.242} C_VEL
LIN {X 0,Y 377.377,Z 417.321,A -85,B 0,C 180,E1 -12292.08,E2 -12292.08} C_VEL
LIN {X 0,Y 377.611,Z 420.342,A -85,B 0,C 180,E1 -12294.108,E2 -12294.108} C_VEL
LIN {X 0,Y 377.254,Z 424.896,A -85,B 0,C 180,E1 -12296.964,E2 -12296.964} C_VEL
LIN {X 0,Y 376.77,Z 429.548,A -85,B 0,C 180,E1 -12299.759,E2 -12299.759} C_VEL
LIN {X 0,Y 376.16,Z 435.776,A -85,B 0,C 180,E1 -12303.359,E2 -12303.359} C_VEL
LIN {X 0,Y 375.711,Z 442.037,A -85,B 0,C 180,E1 -12306.87,E2 -12306.87} C_VEL
LIN {X 0,Y 375.345,Z 448.06,A -85,B 0,C 180,E1 -12310.054,E2 -12310.054} C_VEL
LIN {X 0,Y 378.492,Z 461.387,A -85,B 0,C 180,E1 -12310.723,E2 -12310.723} C_VEL
LIN {X 0,Y 380.485,Z 473.125,A -85,B 0,C 180,E1 -12311.463,E2 -12311.463} C_VEL
LIN {X 0,Y 381.308,Z 482.595,A -85,B 0,C 180,E1 -12312.157,E2 -12312.157} C_VEL
LIN {X 0,Y 380.413,Z 493.886,A -85,B 0,C 180,E1 -12313.084,E2 -12313.084} C_VEL
LIN {X 0,Y 379.221,Z 504.229,A -85,B 0,C 180,E1 -12314.136,E2 -12314.136} C_VEL
LIN {X 0,Y 378.31,Z 513.72,A -85,B 0,C 180,E1 -12315.339,E2 -12315.339} C_VEL
LIN {X 0,Y 377.262,Z 523.183,A -85,B 0,C 180,E1 -12316.809,E2 -12316.809} C_VEL
LIN {X 0,Y 376.168,Z 531.475,A -85,B 0,C 180,E1 -12318.414,E2 -12318.414} C_VEL
LIN {X 0,Y 375.525,Z 538.176,A -85,B 0,C 180,E1 -12320.031,E2 -12320.031} C_VEL
LIN {X 0,Y 374.951,Z 544.35,A -85,B 0,C 180,E1 -12321.919,E2 -12321.919} C_VEL
LIN {X 0,Y 374.592,Z 549.149,A -85,B 0,C 180,E1 -12323.921,E2 -12323.921} C_VEL
LIN {X 0,Y 374.533,Z 552.128,A -85,B 0,C 180,E1 -12325.695,E2 -12325.695} C_VEL
LIN {X 0,Y 374.457,Z 554.262,A -85,B 0,C 180,E1 -12327.849,E2 -12327.849} C_VEL
LIN {X 0,Y 374.517,Z 554.697,A -85,B 0,C 180,E1 -12328.925,E2 -12328.925} C_VEL
LIN {X 0,Y 374.554,Z 554.743,A -85,B 0,C 180,E1 -12330,E2 -12330} C_VEL
LIN {X 0,Y 374.52,Z 554.401,A -85,B 0,C 180,E1 -12331.075,E2 -12331.075} C_VEL
LIN {X 0,Y 374.475,Z 553.669,A -85,B 0,C 180,E1 -12332.151,E2 -12332.151} C_VEL
LIN {X 0,Y 374.465,Z 552.492,A -85,B 0,C 180,E1 -12333.227,E2 -12333.227} C_VEL
LIN {X 0,Y 374.542,Z 549.963,A -85,B 0,C 180,E1 -12334.843,E2 -12334.843} C_VEL
LIN {X 0,Y 374.631,Z 546.409,A -85,B 0,C 180,E1 -12336.462,E2 -12336.462} C_VEL
LIN {X 0,Y 374.892,Z 541.737,A -85,B 0,C 180,E1 -12338.082,E2 -12338.082} C_VEL
LIN {X 0,Y 375.367,Z 534.675,A -85,B 0,C 180,E1 -12339.973,E2 -12339.973} C_VEL
LIN {X 0,Y 375.984,Z 527.02,A -85,B 0,C 180,E1 -12341.592,E2 -12341.592} C_VEL
LIN {X 0,Y 376.73,Z 519.182,A -85,B 0,C 180,E1 -12342.936,E2 -12342.936} C_VEL
LIN {X 0,Y 377.59,Z 508.586,A -85,B 0,C 180,E1 -12344.404,E2 -12344.404} C_VEL
LIN {X 0,Y 378.495,Z 497.633,A -85,B 0,C 180,E1 -12345.619,E2 -12345.619} C_VEL
LIN {X 0,Y 379.33,Z 487.019,A -85,B 0,C 180,E1 -12346.55,E2 -12346.55} C_VEL
LIN {X 0,Y 379.6,Z 479.55,A -85,B 0,C 180,E1 -12347.092,E2 -12347.092} C_VEL
LIN {X 0,Y 377.982,Z 466.504,A -85,B 0,C 180,E1 -12347.92,E2 -12347.92} C_VEL
LIN {X 0,Y 375.914,Z 453.28,A -85,B 0,C 180,E1 -12348.531,E2 -12348.531} C_VEL
LIN {X 0,Y 375.068,Z 448.21,A -85,B 0,C 180,E1 -12348.716,E2 -12348.716} C_VEL
LIN {X 0,Y 375.389,Z 441.936,A -85,B 0,C 180,E1 -12351.989,E2 -12351.989} C_VEL
LIN {X 0,Y 375.776,Z 435.354,A -85,B 0,C 180,E1 -12355.477,E2 -12355.477} C_VEL
LIN {X 0,Y 376.336,Z 427.657,A -85,B 0,C 180,E1 -12359.661,E2 -12359.661} C_VEL
LIN {X 0,Y 376.704,Z 423.246,A -85,B 0,C 180,E1 -12362.12,E2 -12362.12} C_VEL
LIN {X 0,Y 377.133,Z 417.717,A -85,B 0,C 180,E1 -12365.288,E2 -12365.288} C_VEL
LIN {X 0,Y 376.824,Z 413.252,A -85,B 0,C 180,E1 -12367.985,E2 -12367.985} C_VEL
LIN {X 0,Y 376.034,Z 408.648,A -85,B 0,C 180,E1 -12371.004,E2 -12371.004} C_VEL
LIN {X 0,Y 375.976,Z 408.651,A -85,B 0,C 180,E1 -12374.739,E2 -12374.739} C_VEL
LIN {X 0,Y 375.931,Z 408.655,A -85,B 0,C 180,E1 -12378.398,E2 -12378.398} C_VEL
LIN {X 0,Y 375.971,Z 408.65,A -85,B 0,C 180,E1 -12381.728,E2 -12381.728} C_VEL
LIN {X 0,Y 375.975,Z 408.652,A -85,B 0,C 180,E1 -12385.332,E2 -12385.332} C_VEL
LIN {X 0,Y 375.954,Z 408.654,A -85,B 0,C 180,E1 -12388.437,E2 -12388.437} C_VEL
LIN {X 0,Y 375.996,Z 408.647,A -85,B 0,C 180,E1 -12392.141,E2 -12392.141} C_VEL
LIN {X 0,Y 376,Z 408.65,A -85,B 0,C 180,E1 -12394.538,E2 -12394.538} C_VEL
LIN {X 0,Y 375.956,Z 408.653,A -85,B 0,C 180,E1 -12398.045,E2 -12398.045} C_VEL
LIN {X 0,Y 376.001,Z 408.647,A -85,B 0,C 180,E1 -12401.473,E2 -12401.473} C_VEL
LIN {X 0,Y 376.05,Z 408.644,A -85,B 0,C 180,E1 -12404.832,E2 -12404.832} C_VEL
LIN {X 0,Y 376.042,Z 408.644,A -85,B 0,C 180,E1 -12408.136,E2 -12408.136} C_VEL
LIN {X 0,Y 376.25,Z 408.617,A -85,B 0,C 180,E1 -12411.877,E2 -12411.877} C_VEL
LIN {X 0,Y 376.17,Z 408.63,A -85,B 0,C 180,E1 -12414.64,E2 -12414.64} C_VEL
LIN {X 0,Y 376.346,Z 408.605,A -85,B 0,C 180,E1 -12417.859,E2 -12417.859} C_VEL
LIN {X 0,Y 376.482,Z 408.589,A -85,B 0,C 180,E1 -12420,E2 -12420} C_VEL
LIN {X 0,Y 376.185,Z 408.624,A -85,B 0,C 180,E1 -12423.213,E2 -12423.213} C_VEL
LIN {X 0,Y 376.226,Z 408.621,A -85,B 0,C 180,E1 -12426.629,E2 -12426.629} C_VEL
LIN {X 0,Y 376.197,Z 408.624,A -85,B 0,C 180,E1 -12428.595,E2 -12428.595} C_VEL
LIN {X 0,Y 376.047,Z 408.644,A -85,B 0,C 180,E1 -12431.863,E2 -12431.863} C_VEL
LIN {X 0,Y 376.052,Z 408.64,A -85,B 0,C 180,E1 -12435.168,E2 -12435.168} C_VEL
LIN {X 0,Y 376.016,Z 408.646,A -85,B 0,C 180,E1 -12438.526,E2 -12438.526} C_VEL
LIN {X 0,Y 375.956,Z 408.656,A -85,B 0,C 180,E1 -12441.955,E2 -12441.955} C_VEL
LIN {X 0,Y 375.999,Z 408.649,A -85,B 0,C 180,E1 -12445.461,E2 -12445.461} C_VEL
LIN {X 0,Y 375.97,Z 408.65,A -85,B 0,C 180,E1 -12449.079,E2 -12449.079} C_VEL
LIN {X 0,Y 375.951,Z 408.652,A -85,B 0,C 180,E1 -12452.828,E2 -12452.828} C_VEL
LIN {X 0,Y 375.952,Z 408.655,A -85,B 0,C 180,E1 -12455.416,E2 -12455.416} C_VEL
LIN {X 0,Y 375.972,Z 408.65,A -85,B 0,C 180,E1 -12458.272,E2 -12458.272} C_VEL
LIN {X 0,Y 375.984,Z 408.653,A -85,B 0,C 180,E1 -12461.611,E2 -12461.611} C_VEL
LIN {X 0,Y 376.01,Z 408.647,A -85,B 0,C 180,E1 -12465.256,E2 -12465.256} C_VEL
LIN {X 0,Y 375.996,Z 408.649,A -85,B 0,C 180,E1 -12469.142,E2 -12469.142} C_VEL
LIN {X 0,Y 375.964,Z 408.652,A -85,B 0,C 180,E1 -12471.913,E2 -12471.913} C_VEL
LIN {X 0,Y 375.977,Z 408.654,A -85,B 0,C 180,E1 -12475.333,E2 -12475.333} C_VEL
LIN {X 0,Y 375.955,Z 408.651,A -85,B 0,C 180,E1 -12478.439,E2 -12478.439} C_VEL
LIN {X 0,Y 375.994,Z 408.646,A -85,B 0,C 180,E1 -12482.142,E2 -12482.142} C_VEL
LIN {X 0,Y 376.003,Z 408.646,A -85,B 0,C 180,E1 -12484.54,E2 -12484.54} C_VEL
LIN {X 0,Y 375.958,Z 408.654,A -85,B 0,C 180,E1 -12486.887,E2 -12486.887} C_VEL
LIN {X 0,Y 375.777,Z 408.693,A -85,B 0,C 180,E1 -12489.249,E2 -12489.249} C_VEL
LIN {X 0,Y 375.67,Z 412.69,A -85,B 0,C 180,E1 -12492.583,E2 -12492.583} C_VEL
LIN {X 0,Y 375.518,Z 417.765,A -85,B 0,C 180,E1 -12496.706,E2 -12496.706} C_VEL
LIN {X 0,Y 375.271,Z 422.32,A -85,B 0,C 180,E1 -12500.297,E2 -12500.297} C_VEL
LIN {X 0,Y 375.279,Z 426.504,A -85,B 0,C 180,E1 -12503.549,E2 -12503.549} C_VEL
LIN {X 0,Y 375.163,Z 428.885,A -85,B 0,C 180,E1 -12505.367,E2 -12505.367} C_VEL
LIN {X 0,Y 378.101,Z 443.978,A -85,B 0,C 180,E1 -12506.07,E2 -12506.07} C_VEL
LIN {X 0,Y 380.24,Z 455.947,A -85,B 0,C 180,E1 -12506.822,E2 -12506.822} C_VEL
LIN {X 0,Y 379.673,Z 467.112,A -85,B 0,C 180,E1 -12507.624,E2 -12507.624} C_VEL
LIN {X 0,Y 378.791,Z 478.537,A -85,B 0,C 180,E1 -12508.671,E2 -12508.671} C_VEL
LIN {X 0,Y 377.905,Z 488.941,A -85,B 0,C 180,E1 -12509.867,E2 -12509.867} C_VEL
LIN {X 0,Y 377.11,Z 497.462,A -85,B 0,C 180,E1 -12511.068,E2 -12511.068} C_VEL
LIN {X 0,Y 376.379,Z 505.32,A -85,B 0,C 180,E1 -12512.408,E2 -12512.408} C_VEL
LIN {X 0,Y 375.707,Z 512.991,A -85,B 0,C 180,E1 -12514.023,E2 -12514.023} C_VEL
LIN {X 0,Y 375.287,Z 518.247,A -85,B 0,C 180,E1 -12515.373,E2 -12515.373} C_VEL
LIN {X 0,Y 374.995,Z 523.186,A -85,B 0,C 180,E1 -12516.943,E2 -12516.943} C_VEL
LIN {X 0,Y 374.716,Z 527.287,A -85,B 0,C 180,E1 -12518.63,E2 -12518.63} C_VEL
LIN {X 0,Y 374.552,Z 529.328,A -85,B 0,C 180,E1 -12519.722,E2 -12519.722} C_VEL
LIN {X 0,Y 374.465,Z 530.947,A -85,B 0,C 180,E1 -12520.817,E2 -12520.817} C_VEL
LIN {X 0,Y 374.438,Z 532.642,A -85,B 0,C 180,E1 -12522.576,E2 -12522.576} C_VEL
LIN {X 0,Y 374.319,Z 533.245,A -85,B 0,C 180,E1 -12524.127,E2 -12524.127} C_VEL
LIN {X 0,Y 374.324,Z 533.196,A -85,B 0,C 180,E1 -12525.239,E2 -12525.239} C_VEL
LIN {X 0,Y 374.424,Z 532.376,A -85,B 0,C 180,E1 -12526.808,E2 -12526.808} C_VEL
LIN {X 0,Y 374.646,Z 530.429,A -85,B 0,C 180,E1 -12528.596,E2 -12528.596} C_VEL
LIN {X 0,Y 374.995,Z 527.245,A -85,B 0,C 180,E1 -12530.434,E2 -12530.434} C_VEL
LIN {X 0,Y 375.365,Z 523.5,A -85,B 0,C 180,E1 -12531.991,E2 -12531.991} C_VEL
LIN {X 0,Y 376.036,Z 517.492,A -85,B 0,C 180,E1 -12533.894,E2 -12533.894} C_VEL
LIN {X 0,Y 376.881,Z 510.13,A -85,B 0,C 180,E1 -12535.693,E2 -12535.693} C_VEL
LIN {X 0,Y 377.705,Z 503.18,A -85,B 0,C 180,E1 -12537.061,E2 -12537.061} C_VEL
LIN {X 0,Y 378.735,Z 493.993,A -85,B 0,C 180,E1 -12538.543,E2 -12538.543} C_VEL
LIN {X 0,Y 379.663,Z 486.311,A -85,B 0,C 180,E1 -12539.555,E2 -12539.555} C_VEL
LIN {X 0,Y 379.641,Z 481.753,A -85,B 0,C 180,E1 -12540.122,E2 -12540.122} C_VEL
LIN {X 0,Y 377.73,Z 474.213,A -85,B 0,C 180,E1 -12541.053,E2 -12541.053} C_VEL
LIN {X 0,Y 375.68,Z 466.278,A -85,B 0,C 180,E1 -12541.904,E2 -12541.904} C_VEL
LIN {X 0,Y 375.432,Z 461.101,A -85,B 0,C 180,E1 -12542.336,E2 -12542.336} C_VEL
LIN {X 0,Y 375.088,Z 456.696,A -85,B 0,C 180,E1 -12542.681,E2 -12542.681} C_VEL
LIN {X 0,Y 372.612,Z 444.969,A -85,B 0,C 180,E1 -12543.54,E2 -12543.54} C_VEL
LIN {X 0,Y 368.727,Z 431.932,A -85,B 0,C 180,E1 -12544.344,E2 -12544.344} C_VEL
LIN {X 0,Y 368.06,Z 429.445,A -85,B 0,C 180,E1 -12544.501,E2 -12544.501} C_VEL
LIN {X 0,Y 368.291,Z 425.67,A -85,B 0,C 180,E1 -12547.636,E2 -12547.636} C_VEL
LIN {X 0,Y 368.485,Z 422.404,A -85,B 0,C 180,E1 -12550.426,E2 -12550.426} C_VEL
LIN {X 0,Y 368.694,Z 418.815,A -85,B 0,C 180,E1 -12553.585,E2 -12553.585} C_VEL
LIN {X 0,Y 368.954,Z 415.391,A -85,B 0,C 180,E1 -12556.706,E2 -12556.706} C_VEL
LIN {X 0,Y 369.106,Z 412.272,A -85,B 0,C 180,E1 -12559.656,E2 -12559.656} C_VEL
LIN {X 0,Y 368.878,Z 409.542,A -85,B 0,C 180,E1 -12562.434,E2 -12562.434} C_VEL
LIN {X 0,Y 368.932,Z 409.536,A -85,B 0,C 180,E1 -12565.146,E2 -12565.146} C_VEL
LIN {X 0,Y 368.925,Z 409.533,A -85,B 0,C 180,E1 -12569.046,E2 -12569.046} C_VEL
LIN {X 0,Y 368.982,Z 409.525,A -85,B 0,C 180,E1 -12571.564,E2 -12571.564} C_VEL
LIN {X 0,Y 368.995,Z 409.522,A -85,B 0,C 180,E1 -12574.02,E2 -12574.02} C_VEL
LIN {X 0,Y 368.919,Z 409.53,A -85,B 0,C 180,E1 -12577.604,E2 -12577.604} C_VEL
LIN {X 0,Y 368.977,Z 409.523,A -85,B 0,C 180,E1 -12581.107,E2 -12581.107} C_VEL
LIN {X 0,Y 368.992,Z 409.525,A -85,B 0,C 180,E1 -12584.535,E2 -12584.535} C_VEL
LIN {X 0,Y 369,Z 409.521,A -85,B 0,C 180,E1 -12587.907,E2 -12587.907} C_VEL
LIN {X 0,Y 369.224,Z 409.494,A -85,B 0,C 180,E1 -12591.801,E2 -12591.801} C_VEL
LIN {X 0,Y 369.139,Z 409.504,A -85,B 0,C 180,E1 -12594.538,E2 -12594.538} C_VEL
LIN {X 0,Y 369.313,Z 409.483,A -85,B 0,C 180,E1 -12597.819,E2 -12597.819} C_VEL
LIN {X 0,Y 369.452,Z 409.465,A -85,B 0,C 180,E1 -12600,E2 -12600} C_VEL
LIN {X 0,Y 369.314,Z 409.483,A -85,B 0,C 180,E1 -12602.181,E2 -12602.181} C_VEL
LIN {X 0,Y 369.197,Z 409.496,A -85,B 0,C 180,E1 -12606.559,E2 -12606.559} C_VEL
LIN {X 0,Y 369.118,Z 409.508,A -85,B 0,C 180,E1 -12608.762,E2 -12608.762} C_VEL
LIN {X 0,Y 369.009,Z 409.52,A -85,B 0,C 180,E1 -12612.093,E2 -12612.093} C_VEL
LIN {X 0,Y 368.997,Z 409.522,A -85,B 0,C 180,E1 -12615.465,E2 -12615.465} C_VEL
LIN {X 0,Y 368.978,Z 409.527,A -85,B 0,C 180,E1 -12618.893,E2 -12618.893} C_VEL
LIN {X 0,Y 368.928,Z 409.533,A -85,B 0,C 180,E1 -12622.396,E2 -12622.396} C_VEL
LIN {X 0,Y 368.996,Z 409.524,A -85,B 0,C 180,E1 -12625.981,E2 -12625.981} C_VEL
LIN {X 0,Y 368.964,Z 409.526,A -85,B 0,C 180,E1 -12628.814,E2 -12628.814} C_VEL
LIN {X 0,Y 368.896,Z 409.536,A -85,B 0,C 180,E1 -12632.238,E2 -12632.238} C_VEL
LIN {X 0,Y 368.926,Z 409.53,A -85,B 0,C 180,E1 -12635.002,E2 -12635.002} C_VEL
LIN {X 0,Y 368.907,Z 409.529,A -85,B 0,C 180,E1 -12638.641,E2 -12638.641} C_VEL
LIN {X 0,Y 368.879,Z 409.538,A -85,B 0,C 180,E1 -12642.01,E2 -12642.01} C_VEL
LIN {X 0,Y 368.881,Z 409.537,A -85,B 0,C 180,E1 -12645.177,E2 -12645.177} C_VEL
LIN {X 0,Y 369.601,Z 413.419,A -85,B 0,C 180,E1 -12648.278,E2 -12648.278} C_VEL
LIN {X 0,Y 370.228,Z 417.382,A -85,B 0,C 180,E1 -12651.213,E2 -12651.213} C_VEL
LIN {X 0,Y 370.624,Z 421.38,A -85,B 0,C 180,E1 -12653.997,E2 -12653.997} C_VEL
LIN {X 0,Y 370.303,Z 425.466,A -85,B 0,C 180,E1 -12656.625,E2 -12656.625} C_VEL
LIN {X 0,Y 369.674,Z 431.595,A -85,B 0,C 180,E1 -12660.377,E2 -12660.377} C_VEL
LIN {X 0,Y 369,Z 437.816,A -85,B 0,C 180,E1 -12664.02,E2 -12664.02} C_VEL
LIN {X 0,Y 368.554,Z 444.075,A -85,B 0,C 180,E1 -12667.581,E2 -12667.581} C_VEL
LIN {X 0,Y 368.338,Z 447.794,A -85,B 0,C 180,E1 -12669.582,E2 -12669.582} C_VEL
LIN {X 0,Y 371.566,Z 461.125,A -85,B 0,C 180,E1 -12670.275,E2 -12670.275} C_VEL
LIN {X 0,Y 373.743,Z 473.922,A -85,B 0,C 180,E1 -12671.113,E2 -12671.113} C_VEL
LIN {X 0,Y 374.547,Z 483.212,A -85,B 0,C 180,E1 -12671.823,E2 -12671.823} C_VEL
LIN {X 0,Y 373.64,Z 494.33,A -85,B 0,C 180,E1 -12672.768,E2 -12672.768} C_VEL
LIN {X 0,Y 372.288,Z 505.713,A -85,B 0,C 180,E1 -12673.973,E2 -12673.973} C_VEL
LIN {X 0,Y 371.294,Z 515.569,A -85,B 0,C 180,E1 -12675.301,E2 -12675.301} C_VEL
LIN {X 0,Y 370.131,Z 524.778,A -85,B 0,C 180,E1 -12676.829,E2 -12676.829} C_VEL
LIN {X 0,Y 369.063,Z 532.76,A -85,B 0,C 180,E1 -12678.466,E2 -12678.466} C_VEL
LIN {X 0,Y 368.425,Z 539.183,A -85,B 0,C 180,E1 -12680.114,E2 -12680.114} C_VEL
LIN {X 0,Y 367.905,Z 544.302,A -85,B 0,C 180,E1 -12681.763,E2 -12681.763} C_VEL
LIN {X 0,Y 367.567,Z 548.29,A -85,B 0,C 180,E1 -12683.412,E2 -12683.412} C_VEL
LIN {X 0,Y 367.474,Z 550.351,A -85,B 0,C 180,E1 -12684.513,E2 -12684.513} C_VEL
LIN {X 0,Y 367.441,Z 552,A -85,B 0,C 180,E1 -12685.612,E2 -12685.612} C_VEL
LIN {X 0,Y 367.379,Z 553.248,A -85,B 0,C 180,E1 -12686.71,E2 -12686.71} C_VEL
LIN {X 0,Y 367.358,Z 554.087,A -85,B 0,C 180,E1 -12687.807,E2 -12687.807} C_VEL
LIN {X 0,Y 367.417,Z 554.501,A -85,B 0,C 180,E1 -12688.904,E2 -12688.904} C_VEL
LIN {X 0,Y 367.457,Z 554.53,A -85,B 0,C 180,E1 -12690,E2 -12690} C_VEL
LIN {X 0,Y 367.42,Z 554.171,A -85,B 0,C 180,E1 -12691.096,E2 -12691.096} C_VEL
LIN {X 0,Y 367.376,Z 553.412,A -85,B 0,C 180,E1 -12692.192,E2 -12692.192} C_VEL
LIN {X 0,Y 367.383,Z 552.21,A -85,B 0,C 180,E1 -12693.29,E2 -12693.29} C_VEL
LIN {X 0,Y 367.443,Z 549.644,A -85,B 0,C 180,E1 -12694.937,E2 -12694.937} C_VEL
LIN {X 0,Y 367.564,Z 546.051,A -85,B 0,C 180,E1 -12696.587,E2 -12696.587} C_VEL
LIN {X 0,Y 367.848,Z 541.338,A -85,B 0,C 180,E1 -12698.238,E2 -12698.238} C_VEL
LIN {X 0,Y 368.346,Z 534.23,A -85,B 0,C 180,E1 -12700.165,E2 -12700.165} C_VEL
LIN {X 0,Y 369.002,Z 526.51,A -85,B 0,C 180,E1 -12701.814,E2 -12701.814} C_VEL
LIN {X 0,Y 369.747,Z 518.595,A -85,B 0,C 180,E1 -12703.184,E2 -12703.184} C_VEL
LIN {X 0,Y 370.585,Z 508.906,A -85,B 0,C 180,E1 -12704.554,E2 -12704.554} C_VEL
LIN {X 0,Y 371.495,Z 498.173,A -85,B 0,C 180,E1 -12705.78,E2 -12705.78} C_VEL
LIN {X 0,Y 372.359,Z 487.78,A -85,B 0,C 180,E1 -12706.728,E2 -12706.728} C_VEL
LIN {X 0,Y 372.672,Z 480.493,A -85,B 0,C 180,E1 -12707.278,E2 -12707.278} C_VEL
LIN {X 0,Y 371.153,Z 467.94,A -85,B 0,C 180,E1 -12708.112,E2 -12708.112} C_VEL
LIN {X 0,Y 369.204,Z 455.05,A -85,B 0,C 180,E1 -12708.755,E2 -12708.755} C_VEL
LIN {X 0,Y 367.997,Z 448.011,A -85,B 0,C 180,E1 -12709.017,E2 -12709.017} C_VEL
LIN {X 0,Y 368.351,Z 441.62,A -85,B 0,C 180,E1 -12712.432,E2 -12712.432} C_VEL
LIN {X 0,Y 368.76,Z 435.062,A -85,B 0,C 180,E1 -12715.998,E2 -12715.998} C_VEL
LIN {X 0,Y 369.358,Z 427.348,A -85,B 0,C 180,E1 -12720.279,E2 -12720.279} C_VEL
LIN {X 0,Y 369.764,Z 422.189,A -85,B 0,C 180,E1 -12723.248,E2 -12723.248} C_VEL
LIN {X 0,Y 370.097,Z 418.744,A -85,B 0,C 180,E1 -12725.258,E2 -12725.258} C_VEL
LIN {X 0,Y 369.783,Z 414.14,A -85,B 0,C 180,E1 -12728.102,E2 -12728.102} C_VEL
LIN {X 0,Y 368.986,Z 409.526,A -85,B 0,C 180,E1 -12731.169,E2 -12731.169} C_VEL
LIN {X 0,Y 368.951,Z 409.527,A -85,B 0,C 180,E1 -12734.812,E2 -12734.812} C_VEL
LIN {X 0,Y 368.879,Z 409.533,A -85,B 0,C 180,E1 -12738.177,E2 -12738.177} C_VEL
LIN {X 0,Y 368.906,Z 409.533,A -85,B 0,C 180,E1 -12741.359,E2 -12741.359} C_VEL
LIN {X 0,Y 368.932,Z 409.53,A -85,B 0,C 180,E1 -12745.146,E2 -12745.146} C_VEL
LIN {X 0,Y 368.924,Z 409.532,A -85,B 0,C 180,E1 -12749.046,E2 -12749.046} C_VEL
LIN {X 0,Y 368.981,Z 409.521,A -85,B 0,C 180,E1 -12751.564,E2 -12751.564} C_VEL
LIN {X 0,Y 368.951,Z 409.526,A -85,B 0,C 180,E1 -12755.224,E2 -12755.224} C_VEL
LIN {X 0,Y 368.931,Z 409.531,A -85,B 0,C 180,E1 -12758.973,E2 -12758.973} C_VEL
LIN {X 0,Y 368.983,Z 409.523,A -85,B 0,C 180,E1 -12762.257,E2 -12762.257} C_VEL
LIN {X 0,Y 369.029,Z 409.517,A -85,B 0,C 180,E1 -12766.227,E2 -12766.227} C_VEL
LIN {X 0,Y 369.059,Z 409.513,A -85,B 0,C 180,E1 -12770.131,E2 -12770.131} C_VEL
LIN {X 0,Y 369.181,Z 409.5,A -85,B 0,C 180,E1 -12772.342,E2 -12772.342} C_VEL
LIN {X 0,Y 369.142,Z 409.505,A -85,B 0,C 180,E1 -12774.537,E2 -12774.537} C_VEL
LIN {X 0,Y 369.311,Z 409.481,A -85,B 0,C 180,E1 -12777.819,E2 -12777.819} C_VEL
LIN {X 0,Y 369.452,Z 409.465,A -85,B 0,C 180,E1 -12780,E2 -12780} C_VEL
LIN {X 0,Y 369.312,Z 409.484,A -85,B 0,C 180,E1 -12782.181,E2 -12782.181} C_VEL
LIN {X 0,Y 369.196,Z 409.496,A -85,B 0,C 180,E1 -12786.617,E2 -12786.617} C_VEL
LIN {X 0,Y 369.13,Z 409.503,A -85,B 0,C 180,E1 -12788.761,E2 -12788.761} C_VEL
LIN {X 0,Y 369.002,Z 409.522,A -85,B 0,C 180,E1 -12792.093,E2 -12792.093} C_VEL
LIN {X 0,Y 368.991,Z 409.52,A -85,B 0,C 180,E1 -12795.465,E2 -12795.465} C_VEL
LIN {X 0,Y 368.959,Z 409.523,A -85,B 0,C 180,E1 -12798.894,E2 -12798.894} C_VEL
LIN {X 0,Y 368.925,Z 409.53,A -85,B 0,C 180,E1 -12802.395,E2 -12802.395} C_VEL
LIN {X 0,Y 368.993,Z 409.525,A -85,B 0,C 180,E1 -12805.981,E2 -12805.981} C_VEL
LIN {X 0,Y 368.96,Z 409.523,A -85,B 0,C 180,E1 -12808.814,E2 -12808.814} C_VEL
LIN {X 0,Y 368.903,Z 409.532,A -85,B 0,C 180,E1 -12812.237,E2 -12812.237} C_VEL
LIN {X 0,Y 368.923,Z 409.528,A -85,B 0,C 180,E1 -12815.002,E2 -12815.002} C_VEL
LIN {X 0,Y 368.907,Z 409.529,A -85,B 0,C 180,E1 -12818.642,E2 -12818.642} C_VEL
LIN {X 0,Y 368.937,Z 409.528,A -85,B 0,C 180,E1 -12822.021,E2 -12822.021} C_VEL
LIN {X 0,Y 368.985,Z 409.522,A -85,B 0,C 180,E1 -12825.194,E2 -12825.194} C_VEL
LIN {X 0,Y 368.936,Z 409.526,A -85,B 0,C 180,E1 -12828.186,E2 -12828.186} C_VEL
LIN {X 0,Y 368.91,Z 409.534,A -85,B 0,C 180,E1 -12831.359,E2 -12831.359} C_VEL
LIN {X 0,Y 368.933,Z 409.529,A -85,B 0,C 180,E1 -12835.147,E2 -12835.147} C_VEL
LIN {X 0,Y 368.926,Z 409.53,A -85,B 0,C 180,E1 -12839.047,E2 -12839.047} C_VEL
LIN {X 0,Y 368.977,Z 409.524,A -85,B 0,C 180,E1 -12841.565,E2 -12841.565} C_VEL
LIN {X 0,Y 368.998,Z 409.518,A -85,B 0,C 180,E1 -12844.02,E2 -12844.02} C_VEL
LIN {X 0,Y 368.944,Z 409.525,A -85,B 0,C 180,E1 -12846.421,E2 -12846.421} C_VEL
LIN {X 0,Y 368.745,Z 409.686,A -85,B 0,C 180,E1 -12849.341,E2 -12849.341} C_VEL
LIN {X 0,Y 368.617,Z 413.307,A -85,B 0,C 180,E1 -12852.419,E2 -12852.419} C_VEL
LIN {X 0,Y 368.465,Z 418.591,A -85,B 0,C 180,E1 -12856.769,E2 -12856.769} C_VEL
LIN {X 0,Y 368.228,Z 422.764,A -85,B 0,C 180,E1 -12860.109,E2 -12860.109} C_VEL
LIN {X 0,Y 368.215,Z 426.963,A -85,B 0,C 180,E1 -12863.424,E2 -12863.424} C_VEL
LIN {X 0,Y 368.084,Z 429.315,A -85,B 0,C 180,E1 -12865.089,E2 -12865.089} C_VEL
LIN {X 0,Y 370.676,Z 441.704,A -85,B 0,C 180,E1 -12865.651,E2 -12865.651} C_VEL
LIN {X 0,Y 372.857,Z 454.142,A -85,B 0,C 180,E1 -12866.409,E2 -12866.409} C_VEL
LIN {X 0,Y 373.336,Z 459.151,A -85,B 0,C 180,E1 -12866.763,E2 -12866.763} C_VEL
LIN {X 0,Y 372.475,Z 471.041,A -85,B 0,C 180,E1 -12867.689,E2 -12867.689} C_VEL
LIN {X 0,Y 371.605,Z 481.922,A -85,B 0,C 180,E1 -12868.781,E2 -12868.781} C_VEL
LIN {X 0,Y 370.694,Z 491.697,A -85,B 0,C 180,E1 -12870,E2 -12870} C_VEL
LIN {X 0,Y 369.876,Z 500.587,A -85,B 0,C 180,E1 -12871.361,E2 -12871.361} C_VEL
LIN {X 0,Y 369.002,Z 509.287,A -85,B 0,C 180,E1 -12873.002,E2 -12873.002} C_VEL
LIN {X 0,Y 368.381,Z 516.219,A -85,B 0,C 180,E1 -12874.651,E2 -12874.651} C_VEL
LIN {X 0,Y 367.988,Z 522.573,A -85,B 0,C 180,E1 -12876.58,E2 -12876.58} C_VEL
LIN {X 0,Y 367.696,Z 526.757,A -85,B 0,C 180,E1 -12878.242,E2 -12878.242} C_VEL
LIN {X 0,Y 367.431,Z 529.883,A -85,B 0,C 180,E1 -12879.913,E2 -12879.913} C_VEL
LIN {X 0,Y 367.378,Z 531.429,A -85,B 0,C 180,E1 -12881.029,E2 -12881.029} C_VEL
LIN {X 0,Y 367.327,Z 532.871,A -85,B 0,C 180,E1 -12882.638,E2 -12882.638} C_VEL
LIN {X 0,Y 367.218,Z 533.484,A -85,B 0,C 180,E1 -12884.406,E2 -12884.406} C_VEL
LIN {X 0,Y 367.241,Z 533.343,A -85,B 0,C 180,E1 -12885.541,E2 -12885.541} C_VEL
LIN {X 0,Y 367.348,Z 532.564,A -85,B 0,C 180,E1 -12886.945,E2 -12886.945} C_VEL
LIN {X 0,Y 367.606,Z 530.338,A -85,B 0,C 180,E1 -12888.966,E2 -12888.966} C_VEL
LIN {X 0,Y 367.95,Z 527.437,A -85,B 0,C 180,E1 -12890.623,E2 -12890.623} C_VEL
LIN {X 0,Y 368.408,Z 523.1,A -85,B 0,C 180,E1 -12892.428,E2 -12892.428} C_VEL
LIN {X 0,Y 369.118,Z 517.463,A -85,B 0,C 180,E1 -12894.206,E2 -12894.206} C_VEL
LIN {X 0,Y 369.931,Z 510.63,A -85,B 0,C 180,E1 -12895.91,E2 -12895.91} C_VEL
LIN {X 0,Y 370.851,Z 503.439,A -85,B 0,C 180,E1 -12897.358,E2 -12897.358} C_VEL
LIN {X 0,Y 371.89,Z 494.667,A -85,B 0,C 180,E1 -12898.809,E2 -12898.809} C_VEL
LIN {X 0,Y 373.139,Z 484.553,A -85,B 0,C 180,E1 -12900.145,E2 -12900.145} C_VEL
LIN {X 0,Y 374.229,Z 474.176,A -85,B 0,C 180,E1 -12901.251,E2 -12901.251} C_VEL
LIN {X 0,Y 375.336,Z 462.465,A -85,B 0,C 180,E1 -12902.238,E2 -12902.238} C_VEL
LIN {X 0,Y 375.432,Z 461.101,A -85,B 0,C 180,E1 -12902.336,E2 -12902.336} C_VEL
LIN {X 0,Y 375.163,Z 457.664,A -85,B 0,C 180,E1 -12902.609,E2 -12902.609} C_VEL
LIN {X 0,Y 374.08,Z 454.436,A -85,B 0,C 180,E1 -12902.902,E2 -12902.902} C_VEL
LIN {X 0,Y 370.476,Z 448.518,A -85,B 0,C 180,E1 -12903.503,E2 -12903.503} C_VEL
LIN {X 0,Y 365.247,Z 441.07,A -85,B 0,C 180,E1 -12904.237,E2 -12904.237} C_VEL
LIN {X 0,Y 362.963,Z 435.967,A -85,B 0,C 180,E1 -12904.615,E2 -12904.615} C_VEL
LIN {X 0,Y 361.024,Z 429.669,A -85,B 0,C 180,E1 -12904.982,E2 -12904.982} C_VEL
LIN {X 0,Y 361.305,Z 425.542,A -85,B 0,C 180,E1 -12908.495,E2 -12908.495} C_VEL
LIN {X 0,Y 361.583,Z 421.133,A -85,B 0,C 180,E1 -12912.388,E2 -12912.388} C_VEL
LIN {X 0,Y 361.854,Z 417.26,A -85,B 0,C 180,E1 -12915.94,E2 -12915.94} C_VEL
LIN {X 0,Y 362.053,Z 413.841,A -85,B 0,C 180,E1 -12919.204,E2 -12919.204} C_VEL
LIN {X 0,Y 361.954,Z 411.482,A -85,B 0,C 180,E1 -12921.586,E2 -12921.586} C_VEL
LIN {X 0,Y 361.855,Z 410.418,A -85,B 0,C 180,E1 -12922.981,E2 -12922.981} C_VEL
LIN {X 0,Y 361.858,Z 410.417,A -85,B 0,C 180,E1 -12926.63,E2 -12926.63} C_VEL
LIN {X 0,Y 361.872,Z 410.411,A -85,B 0,C 180,E1 -12929.672,E2 -12929.672} C_VEL
LIN {X 0,Y 361.95,Z 410.4,A -85,B 0,C 180,E1 -12933.475,E2 -12933.475} C_VEL
LIN {X 0,Y 361.877,Z 410.411,A -85,B 0,C 180,E1 -12937.144,E2 -12937.144} C_VEL
LIN {X 0,Y 361.915,Z 410.402,A -85,B 0,C 180,E1 -12940.724,E2 -12940.724} C_VEL
LIN {X 0,Y 361.94,Z 410.401,A -85,B 0,C 180,E1 -12944.226,E2 -12944.226} C_VEL
LIN {X 0,Y 361.993,Z 410.394,A -85,B 0,C 180,E1 -12946.528,E2 -12946.528} C_VEL
LIN {X 0,Y 362.026,Z 410.388,A -85,B 0,C 180,E1 -12949.938,E2 -12949.938} C_VEL
LIN {X 0,Y 362.146,Z 410.377,A -85,B 0,C 180,E1 -12952.193,E2 -12952.193} C_VEL
LIN {X 0,Y 362.112,Z 410.379,A -85,B 0,C 180,E1 -12954.431,E2 -12954.431} C_VEL
LIN {X 0,Y 362.277,Z 410.359,A -85,B 0,C 180,E1 -12957.777,E2 -12957.777} C_VEL
LIN {X 0,Y 362.422,Z 410.341,A -85,B 0,C 180,E1 -12960,E2 -12960} C_VEL
LIN {X 0,Y 362.278,Z 410.36,A -85,B 0,C 180,E1 -12962.224,E2 -12962.224} C_VEL
LIN {X 0,Y 362.159,Z 410.373,A -85,B 0,C 180,E1 -12966.687,E2 -12966.687} C_VEL
LIN {X 0,Y 362.031,Z 410.39,A -85,B 0,C 180,E1 -12970.062,E2 -12970.062} C_VEL
LIN {X 0,Y 361.994,Z 410.393,A -85,B 0,C 180,E1 -12973.9,E2 -12973.9} C_VEL
LIN {X 0,Y 361.963,Z 410.4,A -85,B 0,C 180,E1 -12977.939,E2 -12977.939} C_VEL
LIN {X 0,Y 361.888,Z 410.411,A -85,B 0,C 180,E1 -12981.653,E2 -12981.653} C_VEL
LIN {X 0,Y 361.924,Z 410.405,A -85,B 0,C 180,E1 -12985.291,E2 -12985.291} C_VEL
LIN {X 0,Y 361.919,Z 410.407,A -85,B 0,C 180,E1 -12987.778,E2 -12987.778} C_VEL
LIN {X 0,Y 361.844,Z 410.414,A -85,B 0,C 180,E1 -12991.286,E2 -12991.286} C_VEL
LIN {X 0,Y 361.851,Z 410.412,A -85,B 0,C 180,E1 -12994.281,E2 -12994.281} C_VEL
LIN {X 0,Y 361.862,Z 410.406,A -85,B 0,C 180,E1 -12997.224,E2 -12997.224} C_VEL
LIN {X 0,Y 361.833,Z 410.414,A -85,B 0,C 180,E1 -13000.756,E2 -13000.756} C_VEL
LIN {X 0,Y 361.816,Z 410.416,A -85,B 0,C 180,E1 -13004.369,E2 -13004.369} C_VEL
LIN {X 0,Y 361.913,Z 410.799,A -85,B 0,C 180,E1 -13005.021,E2 -13005.021} C_VEL
LIN {X 0,Y 362.742,Z 415.462,A -85,B 0,C 180,E1 -13008.797,E2 -13008.797} C_VEL
LIN {X 0,Y 363.315,Z 419.424,A -85,B 0,C 180,E1 -13011.757,E2 -13011.757} C_VEL
LIN {X 0,Y 363.627,Z 422.997,A -85,B 0,C 180,E1 -13014.268,E2 -13014.268} C_VEL
LIN {X 0,Y 363.178,Z 427.499,A -85,B 0,C 180,E1 -13017.192,E2 -13017.192} C_VEL
LIN {X 0,Y 362.56,Z 433.182,A -85,B 0,C 180,E1 -13020.727,E2 -13020.727} C_VEL
LIN {X 0,Y 361.855,Z 439.849,A -85,B 0,C 180,E1 -13024.705,E2 -13024.705} C_VEL
LIN {X 0,Y 361.422,Z 446.112,A -85,B 0,C 180,E1 -13028.318,E2 -13028.318} C_VEL
LIN {X 0,Y 361.338,Z 447.446,A -85,B 0,C 180,E1 -13029.077,E2 -13029.077} C_VEL
LIN {X 0,Y 364.615,Z 461.089,A -85,B 0,C 180,E1 -13029.815,E2 -13029.815} C_VEL
LIN {X 0,Y 366.805,Z 473.014,A -85,B 0,C 180,E1 -13030.623,E2 -13030.623} C_VEL
LIN {X 0,Y 367.796,Z 483.837,A -85,B 0,C 180,E1 -13031.478,E2 -13031.478} C_VEL
LIN {X 0,Y 367.062,Z 493.376,A -85,B 0,C 180,E1 -13032.305,E2 -13032.305} C_VEL
LIN {X 0,Y 365.612,Z 504.892,A -85,B 0,C 180,E1 -13033.529,E2 -13033.529} C_VEL
LIN {X 0,Y 364.579,Z 514.03,A -85,B 0,C 180,E1 -13034.75,E2 -13034.75} C_VEL
LIN {X 0,Y 363.409,Z 523.44,A -85,B 0,C 180,E1 -13036.296,E2 -13036.296} C_VEL
LIN {X 0,Y 362.25,Z 531.609,A -85,B 0,C 180,E1 -13037.962,E2 -13037.962} C_VEL
LIN {X 0,Y 361.615,Z 537.198,A -85,B 0,C 180,E1 -13039.36,E2 -13039.36} C_VEL
LIN {X 0,Y 361.039,Z 542.675,A -85,B 0,C 180,E1 -13041.041,E2 -13041.041} C_VEL
LIN {X 0,Y 360.607,Z 546.983,A -85,B 0,C 180,E1 -13042.722,E2 -13042.722} C_VEL
LIN {X 0,Y 360.394,Z 550.241,A -85,B 0,C 180,E1 -13044.404,E2 -13044.404} C_VEL
LIN {X 0,Y 360.352,Z 551.871,A -85,B 0,C 180,E1 -13045.526,E2 -13045.526} C_VEL
LIN {X 0,Y 360.298,Z 553.103,A -85,B 0,C 180,E1 -13046.645,E2 -13046.645} C_VEL
LIN {X 0,Y 360.263,Z 553.907,A -85,B 0,C 180,E1 -13047.764,E2 -13047.764} C_VEL
LIN {X 0,Y 360.317,Z 554.304,A -85,B 0,C 180,E1 -13048.882,E2 -13048.882} C_VEL
LIN {X 0,Y 360.36,Z 554.316,A -85,B 0,C 180,E1 -13050,E2 -13050} C_VEL
LIN {X 0,Y 360.321,Z 553.941,A -85,B 0,C 180,E1 -13051.117,E2 -13051.117} C_VEL
LIN {X 0,Y 360.279,Z 553.15,A -85,B 0,C 180,E1 -13052.236,E2 -13052.236} C_VEL
LIN {X 0,Y 360.303,Z 551.929,A -85,B 0,C 180,E1 -13053.354,E2 -13053.354} C_VEL
LIN {X 0,Y 360.347,Z 549.324,A -85,B 0,C 180,E1 -13055.035,E2 -13055.035} C_VEL
LIN {X 0,Y 360.498,Z 545.694,A -85,B 0,C 180,E1 -13056.717,E2 -13056.717} C_VEL
LIN {X 0,Y 360.796,Z 540.939,A -85,B 0,C 180,E1 -13058.4,E2 -13058.4} C_VEL
LIN {X 0,Y 361.332,Z 533.785,A -85,B 0,C 180,E1 -13060.364,E2 -13060.364} C_VEL
LIN {X 0,Y 362.022,Z 525.988,A -85,B 0,C 180,E1 -13062.045,E2 -13062.045} C_VEL
LIN {X 0,Y 362.771,Z 518,A -85,B 0,C 180,E1 -13063.442,E2 -13063.442} C_VEL
LIN {X 0,Y 363.651,Z 508.216,A -85,B 0,C 180,E1 -13064.84,E2 -13064.84} C_VEL
LIN {X 0,Y 364.599,Z 497.386,A -85,B 0,C 180,E1 -13066.086,E2 -13066.086} C_VEL
LIN {X 0,Y 365.543,Z 486.827,A -85,B 0,C 180,E1 -13067.049,E2 -13067.049} C_VEL
LIN {X 0,Y 365.633,Z 480.355,A -85,B 0,C 180,E1 -13067.549,E2 -13067.549} C_VEL
LIN {X 0,Y 364.126,Z 467.825,A -85,B 0,C 180,E1 -13068.398,E2 -13068.398} C_VEL
LIN {X 0,Y 362.102,Z 454.631,A -85,B 0,C 180,E1 -13069.071,E2 -13069.071} C_VEL
LIN {X 0,Y 360.934,Z 447.836,A -85,B 0,C 180,E1 -13069.33,E2 -13069.33} C_VEL
LIN {X 0,Y 361.317,Z 441.309,A -85,B 0,C 180,E1 -13072.893,E2 -13072.893} C_VEL
LIN {X 0,Y 361.687,Z 435.828,A -85,B 0,C 180,E1 -13075.925,E2 -13075.925} C_VEL
LIN {X 0,Y 362.297,Z 428.16,A -85,B 0,C 180,E1 -13080.288,E2 -13080.288} C_VEL
LIN {X 0,Y 362.668,Z 423.746,A -85,B 0,C 180,E1 -13082.86,E2 -13082.86} C_VEL
LIN {X 0,Y 363.061,Z 419.147,A -85,B 0,C 180,E1 -13085.607,E2 -13085.607} C_VEL
LIN {X 0,Y 362.72,Z 414.864,A -85,B 0,C 180,E1 -13088.317,E2 -13088.317} C_VEL
LIN {X 0,Y 361.941,Z 410.403,A -85,B 0,C 180,E1 -13091.314,E2 -13091.314} C_VEL
LIN {X 0,Y 361.901,Z 410.402,A -85,B 0,C 180,E1 -13094.354,E2 -13094.354} C_VEL
LIN {X 0,Y 361.833,Z 410.412,A -85,B 0,C 180,E1 -13097.567,E2 -13097.567} C_VEL
LIN {X 0,Y 361.867,Z 410.412,A -85,B 0,C 180,E1 -13100.972,E2 -13100.972} C_VEL
LIN {X 0,Y 361.87,Z 410.409,A -85,B 0,C 180,E1 -13104.654,E2 -13104.654} C_VEL
LIN {X 0,Y 361.833,Z 410.412,A -85,B 0,C 180,E1 -13108.37,E2 -13108.37} C_VEL
LIN {X 0,Y 361.897,Z 410.407,A -85,B 0,C 180,E1 -13110.955,E2 -13110.955} C_VEL
LIN {X 0,Y 361.949,Z 410.397,A -85,B 0,C 180,E1 -13113.474,E2 -13113.474} C_VEL
LIN {X 0,Y 361.883,Z 410.407,A -85,B 0,C 180,E1 -13117.144,E2 -13117.144} C_VEL
LIN {X 0,Y 361.899,Z 410.407,A -85,B 0,C 180,E1 -13120.723,E2 -13120.723} C_VEL
LIN {X 0,Y 361.925,Z 410.402,A -85,B 0,C 180,E1 -13123.065,E2 -13123.065} C_VEL
LIN {X 0,Y 361.991,Z 410.396,A -85,B 0,C 180,E1 -13126.527,E2 -13126.527} C_VEL
LIN {X 0,Y 362.023,Z 410.388,A -85,B 0,C 180,E1 -13129.938,E2 -13129.938} C_VEL
LIN {X 0,Y 362.139,Z 410.376,A -85,B 0,C 180,E1 -13132.192,E2 -13132.192} C_VEL
LIN {X 0,Y 362.115,Z 410.38,A -85,B 0,C 180,E1 -13134.431,E2 -13134.431} C_VEL
LIN {X 0,Y 362.275,Z 410.357,A -85,B 0,C 180,E1 -13137.776,E2 -13137.776} C_VEL
LIN {X 0,Y 362.421,Z 410.34,A -85,B 0,C 180,E1 -13140,E2 -13140} C_VEL
LIN {X 0,Y 362.276,Z 410.36,A -85,B 0,C 180,E1 -13142.223,E2 -13142.223} C_VEL
LIN {X 0,Y 362.164,Z 410.372,A -85,B 0,C 180,E1 -13146.686,E2 -13146.686} C_VEL
LIN {X 0,Y 362.066,Z 410.382,A -85,B 0,C 180,E1 -13148.933,E2 -13148.933} C_VEL
LIN {X 0,Y 361.956,Z 410.4,A -85,B 0,C 180,E1 -13152.332,E2 -13152.332} C_VEL
LIN {X 0,Y 361.955,Z 410.397,A -85,B 0,C 180,E1 -13154.62,E2 -13154.62} C_VEL
LIN {X 0,Y 361.95,Z 410.402,A -85,B 0,C 180,E1 -13158.1,E2 -13158.1} C_VEL
LIN {X 0,Y 361.884,Z 410.407,A -85,B 0,C 180,E1 -13161.653,E2 -13161.653} C_VEL
LIN {X 0,Y 361.921,Z 410.401,A -85,B 0,C 180,E1 -13165.29,E2 -13165.29} C_VEL
LIN {X 0,Y 361.916,Z 410.405,A -85,B 0,C 180,E1 -13167.778,E2 -13167.778} C_VEL
LIN {X 0,Y 361.853,Z 410.412,A -85,B 0,C 180,E1 -13171.628,E2 -13171.628} C_VEL
LIN {X 0,Y 361.868,Z 410.409,A -85,B 0,C 180,E1 -13175.345,E2 -13175.345} C_VEL
LIN {X 0,Y 361.869,Z 410.407,A -85,B 0,C 180,E1 -13179.028,E2 -13179.028} C_VEL
LIN {X 0,Y 361.882,Z 410.404,A -85,B 0,C 180,E1 -13182.441,E2 -13182.441} C_VEL
LIN {X 0,Y 361.924,Z 410.401,A -85,B 0,C 180,E1 -13185.929,E2 -13185.929} C_VEL
LIN {X 0,Y 361.901,Z 410.405,A -85,B 0,C 180,E1 -13189.232,E2 -13189.232} C_VEL
LIN {X 0,Y 361.866,Z 410.408,A -85,B 0,C 180,E1 -13192.983,E2 -13192.983} C_VEL
LIN {X 0,Y 361.855,Z 410.408,A -85,B 0,C 180,E1 -13196.631,E2 -13196.631} C_VEL
LIN {X 0,Y 361.872,Z 410.408,A -85,B 0,C 180,E1 -13199.673,E2 -13199.673} C_VEL
LIN {X 0,Y 361.953,Z 410.399,A -85,B 0,C 180,E1 -13203.476,E2 -13203.476} C_VEL
LIN {X 0,Y 361.903,Z 410.402,A -85,B 0,C 180,E1 -13205.933,E2 -13205.933} C_VEL
LIN {X 0,Y 361.696,Z 410.591,A -85,B 0,C 180,E1 -13209.359,E2 -13209.359} C_VEL
LIN {X 0,Y 361.515,Z 414.89,A -85,B 0,C 180,E1 -13213.046,E2 -13213.046} C_VEL
LIN {X 0,Y 361.416,Z 419.022,A -85,B 0,C 180,E1 -13216.506,E2 -13216.506} C_VEL
LIN {X 0,Y 361.154,Z 423.203,A -85,B 0,C 180,E1 -13219.914,E2 -13219.914} C_VEL
LIN {X 0,Y 361.16,Z 427.431,A -85,B 0,C 180,E1 -13223.295,E2 -13223.295} C_VEL
LIN {X 0,Y 360.991,Z 429.298,A -85,B 0,C 180,E1 -13224.764,E2 -13224.764} C_VEL
LIN {X 0,Y 363.742,Z 442.324,A -85,B 0,C 180,E1 -13225.377,E2 -13225.377} C_VEL
LIN {X 0,Y 365.982,Z 455.404,A -85,B 0,C 180,E1 -13226.202,E2 -13226.202} C_VEL
LIN {X 0,Y 366.388,Z 460.759,A -85,B 0,C 180,E1 -13226.593,E2 -13226.593} C_VEL
LIN {X 0,Y 365.531,Z 471.862,A -85,B 0,C 180,E1 -13227.493,E2 -13227.493} C_VEL
LIN {X 0,Y 364.62,Z 482.723,A -85,B 0,C 180,E1 -13228.62,E2 -13228.62} C_VEL
LIN {X 0,Y 363.592,Z 493.377,A -85,B 0,C 180,E1 -13230,E2 -13230} C_VEL
LIN {X 0,Y 362.756,Z 502.028,A -85,B 0,C 180,E1 -13231.388,E2 -13231.388} C_VEL
LIN {X 0,Y 361.867,Z 510.438,A -85,B 0,C 180,E1 -13233.062,E2 -13233.062} C_VEL
LIN {X 0,Y 361.243,Z 517.199,A -85,B 0,C 180,E1 -13234.743,E2 -13234.743} C_VEL
LIN {X 0,Y 360.862,Z 523.397,A -85,B 0,C 180,E1 -13236.711,E2 -13236.711} C_VEL
LIN {X 0,Y 360.576,Z 527.439,A -85,B 0,C 180,E1 -13238.406,E2 -13238.406} C_VEL
LIN {X 0,Y 360.316,Z 530.435,A -85,B 0,C 180,E1 -13240.11,E2 -13240.11} C_VEL
LIN {X 0,Y 360.279,Z 531.861,A -85,B 0,C 180,E1 -13241.249,E2 -13241.249} C_VEL
LIN {X 0,Y 360.237,Z 533.11,A -85,B 0,C 180,E1 -13242.718,E2 -13242.718} C_VEL
LIN {X 0,Y 360.124,Z 533.702,A -85,B 0,C 180,E1 -13244.697,E2 -13244.697} C_VEL
LIN {X 0,Y 360.176,Z 533.455,A -85,B 0,C 180,E1 -13245.853,E2 -13245.853} C_VEL
LIN {X 0,Y 360.273,Z 532.754,A -85,B 0,C 180,E1 -13247.087,E2 -13247.087} C_VEL
LIN {X 0,Y 360.416,Z 531.744,A -85,B 0,C 180,E1 -13248.179,E2 -13248.179} C_VEL
LIN {X 0,Y 360.71,Z 529.276,A -85,B 0,C 180,E1 -13249.936,E2 -13249.936} C_VEL
LIN {X 0,Y 361.128,Z 525.725,A -85,B 0,C 180,E1 -13251.701,E2 -13251.701} C_VEL
LIN {X 0,Y 361.716,Z 520.961,A -85,B 0,C 180,E1 -13253.472,E2 -13253.472} C_VEL
LIN {X 0,Y 362.52,Z 514.813,A -85,B 0,C 180,E1 -13255.246,E2 -13255.246} C_VEL
LIN {X 0,Y 363.472,Z 507.851,A -85,B 0,C 180,E1 -13256.852,E2 -13256.852} C_VEL
LIN {X 0,Y 364.589,Z 499.045,A -85,B 0,C 180,E1 -13258.495,E2 -13258.495} C_VEL
LIN {X 0,Y 365.908,Z 489.153,A -85,B 0,C 180,E1 -13259.959,E2 -13259.959} C_VEL
LIN {X 0,Y 367.204,Z 478.016,A -85,B 0,C 180,E1 -13261.275,E2 -13261.275} C_VEL
LIN {X 0,Y 368.353,Z 467.14,A -85,B 0,C 180,E1 -13262.291,E2 -13262.291} C_VEL
LIN {X 0,Y 368.813,Z 460.565,A -85,B 0,C 180,E1 -13262.801,E2 -13262.801} C_VEL
LIN {X 0,Y 366.703,Z 449.417,A -85,B 0,C 180,E1 -13263.695,E2 -13263.695} C_VEL
LIN {X 0,Y 363.39,Z 437.265,A -85,B 0,C 180,E1 -13264.53,E2 -13264.53} C_VEL
LIN {X 0,Y 362.963,Z 435.967,A -85,B 0,C 180,E1 -13264.615,E2 -13264.615} C_VEL
LIN {X 0,Y 361.759,Z 433.024,A -85,B 0,C 180,E1 -13264.922,E2 -13264.922} C_VEL
LIN {X 0,Y 360.325,Z 430.883,A -85,B 0,C 180,E1 -13265.36,E2 -13265.36} C_VEL
LIN {X 0,Y 358.126,Z 428.823,A -85,B 0,C 180,E1 -13266.163,E2 -13266.163} C_VEL
LIN {X 0,Y 355.131,Z 427.172,A -85,B 0,C 180,E1 -13267.755,E2 -13267.755} C_VEL
LIN {X 0,Y 354.308,Z 426.137,A -85,B 0,C 180,E1 -13268.769,E2 -13268.769} C_VEL
LIN {X 0,Y 354.281,Z 425.752,A -85,B 0,C 180,E1 -13269.109,E2 -13269.109} C_VEL
LIN {X 0,Y 354.564,Z 422.118,A -85,B 0,C 180,E1 -13272.371,E2 -13272.371} C_VEL
LIN {X 0,Y 354.859,Z 418.115,A -85,B 0,C 180,E1 -13276.118,E2 -13276.118} C_VEL
LIN {X 0,Y 355.046,Z 414.948,A -85,B 0,C 180,E1 -13279.215,E2 -13279.215} C_VEL
LIN {X 0,Y 354.879,Z 411.881,A -85,B 0,C 180,E1 -13282.386,E2 -13282.386} C_VEL
LIN {X 0,Y 354.789,Z 411.298,A -85,B 0,C 180,E1 -13283.54,E2 -13283.54} C_VEL
LIN {X 0,Y 354.827,Z 411.292,A -85,B 0,C 180,E1 -13286.318,E2 -13286.318} C_VEL
LIN {X 0,Y 354.85,Z 411.285,A -85,B 0,C 180,E1 -13290.321,E2 -13290.321} C_VEL
LIN {X 0,Y 354.894,Z 411.279,A -85,B 0,C 180,E1 -13294.172,E2 -13294.172} C_VEL
LIN {X 0,Y 354.812,Z 411.287,A -85,B 0,C 180,E1 -13297.893,E2 -13297.893} C_VEL
LIN {X 0,Y 354.918,Z 411.276,A -85,B 0,C 180,E1 -13301.891,E2 -13301.891} C_VEL
LIN {X 0,Y 354.937,Z 411.27,A -85,B 0,C 180,E1 -13305.981,E2 -13305.981} C_VEL
LIN {X 0,Y 354.973,Z 411.267,A -85,B 0,C 180,E1 -13309.736,E2 -13309.736} C_VEL
LIN {X 0,Y 355.109,Z 411.253,A -85,B 0,C 180,E1 -13312.037,E2 -13312.037} C_VEL
LIN {X 0,Y 355.087,Z 411.254,A -85,B 0,C 180,E1 -13314.321,E2 -13314.321} C_VEL
LIN {X 0,Y 355.24,Z 411.235,A -85,B 0,C 180,E1 -13317.733,E2 -13317.733} C_VEL
LIN {X 0,Y 355.392,Z 411.217,A -85,B 0,C 180,E1 -13320,E2 -13320} C_VEL
LIN {X 0,Y 355.241,Z 411.236,A -85,B 0,C 180,E1 -13322.268,E2 -13322.268} C_VEL
LIN {X 0,Y 355.123,Z 411.247,A -85,B 0,C 180,E1 -13326.82,E2 -13326.82} C_VEL
LIN {X 0,Y 354.978,Z 411.268,A -85,B 0,C 180,E1 -13330.264,E2 -13330.264} C_VEL
LIN {X 0,Y 354.939,Z 411.272,A -85,B 0,C 180,E1 -13334.02,E2 -13334.02} C_VEL
LIN {X 0,Y 354.919,Z 411.277,A -85,B 0,C 180,E1 -13338.109,E2 -13338.109} C_VEL
LIN {X 0,Y 354.83,Z 411.289,A -85,B 0,C 180,E1 -13342.107,E2 -13342.107} C_VEL
LIN {X 0,Y 354.896,Z 411.28,A -85,B 0,C 180,E1 -13345.828,E2 -13345.828} C_VEL
LIN {X 0,Y 354.851,Z 411.285,A -85,B 0,C 180,E1 -13349.679,E2 -13349.679} C_VEL
LIN {X 0,Y 354.803,Z 411.291,A -85,B 0,C 180,E1 -13353.703,E2 -13353.703} C_VEL
LIN {X 0,Y 354.796,Z 411.287,A -85,B 0,C 180,E1 -13356.46,E2 -13356.46} C_VEL
LIN {X 0,Y 354.822,Z 411.284,A -85,B 0,C 180,E1 -13359.424,E2 -13359.424} C_VEL
LIN {X 0,Y 354.786,Z 411.292,A -85,B 0,C 180,E1 -13362.868,E2 -13362.868} C_VEL
LIN {X 0,Y 354.796,Z 411.312,A -85,B 0,C 180,E1 -13364.211,E2 -13364.211} C_VEL
LIN {X 0,Y 355.56,Z 415.552,A -85,B 0,C 180,E1 -13367.776,E2 -13367.776} C_VEL
LIN {X 0,Y 356.187,Z 419.465,A -85,B 0,C 180,E1 -13370.847,E2 -13370.847} C_VEL
LIN {X 0,Y 356.614,Z 423.669,A -85,B 0,C 180,E1 -13373.902,E2 -13373.902} C_VEL
LIN {X 0,Y 356.278,Z 427.503,A -85,B 0,C 180,E1 -13376.473,E2 -13376.473} C_VEL
LIN {X 0,Y 355.718,Z 432.598,A -85,B 0,C 180,E1 -13379.748,E2 -13379.748} C_VEL
